LIN {X 0,Y 244.546,Z 349.21,A -85,B 0,C 180,E1 -19754.66,E2 -19754.66} C_VEL
LIN {X 0,Y 242.026,Z 345.394,A -85,B 0,C 180,E1 -19755.456,E2 -19755.456} C_VEL
LIN {X 0,Y 239.218,Z 341.212,A -85,B 0,C 180,E1 -19756.337,E2 -19756.337} C_VEL
LIN {X 0,Y 238.833,Z 340.13,A -85,B 0,C 180,E1 -19756.54,E2 -19756.54} C_VEL
LIN {X 0,Y 238.266,Z 336.796,A -85,B 0,C 180,E1 -19760.076,E2 -19760.076} C_VEL
LIN {X 0,Y 237.671,Z 333.533,A -85,B 0,C 180,E1 -19763.743,E2 -19763.743} C_VEL
LIN {X 0,Y 237.026,Z 330.381,A -85,B 0,C 180,E1 -19767.743,E2 -19767.743} C_VEL
LIN {X 0,Y 236.378,Z 327.428,A -85,B 0,C 180,E1 -19771.594,E2 -19771.594} C_VEL
LIN {X 0,Y 235.759,Z 324.904,A -85,B 0,C 180,E1 -19775.333,E2 -19775.333} C_VEL
LIN {X 0,Y 235.115,Z 322.576,A -85,B 0,C 180,E1 -19778.979,E2 -19778.979} C_VEL
LIN {X 0,Y 234.966,Z 321.838,A -85,B 0,C 180,E1 -19780.336,E2 -19780.336} C_VEL
LIN {X 0,Y 235.086,Z 321.809,A -85,B 0,C 180,E1 -19784.392,E2 -19784.392} C_VEL
LIN {X 0,Y 235.285,Z 321.791,A -85,B 0,C 180,E1 -19790.302,E2 -19790.302} C_VEL
LIN {X 0,Y 235.355,Z 321.768,A -85,B 0,C 180,E1 -19793.14,E2 -19793.14} C_VEL
LIN {X 0,Y 235.594,Z 321.742,A -85,B 0,C 180,E1 -19798.29,E2 -19798.29} C_VEL
LIN {X 0,Y 235.59,Z 321.753,A -85,B 0,C 180,E1 -19801.709,E2 -19801.709} C_VEL
LIN {X 0,Y 235.36,Z 321.774,A -85,B 0,C 180,E1 -19806.86,E2 -19806.86} C_VEL
LIN {X 0,Y 235.213,Z 321.785,A -85,B 0,C 180,E1 -19810.327,E2 -19810.327} C_VEL
LIN {X 0,Y 235.114,Z 321.8,A -85,B 0,C 180,E1 -19815.606,E2 -19815.606} C_VEL
LIN {X 0,Y 235.008,Z 321.838,A -85,B 0,C 180,E1 -19819.205,E2 -19819.205} C_VEL
LIN {X 0,Y 234.981,Z 321.816,A -85,B 0,C 180,E1 -19821.415,E2 -19821.415} C_VEL
LIN {X 0,Y 236.066,Z 324.801,A -85,B 0,C 180,E1 -19824.632,E2 -19824.632} C_VEL
LIN {X 0,Y 237.859,Z 328.745,A -85,B 0,C 180,E1 -19828.213,E2 -19828.213} C_VEL
LIN {X 0,Y 239.119,Z 334.547,A -85,B 0,C 180,E1 -19831.941,E2 -19831.941} C_VEL
LIN {X 0,Y 240.693,Z 341.686,A -85,B 0,C 180,E1 -19835.731,E2 -19835.731} C_VEL
LIN {X 0,Y 241.887,Z 346.106,A -85,B 0,C 180,E1 -19837.864,E2 -19837.864} C_VEL
LIN {X 0,Y 241.737,Z 348.256,A -85,B 0,C 180,E1 -19838.655,E2 -19838.655} C_VEL
LIN {X 0,Y 239.964,Z 352.557,A -85,B 0,C 180,E1 -19839.813,E2 -19839.813} C_VEL
LIN {X 0,Y 238.2,Z 356.932,A -85,B 0,C 180,E1 -19840.981,E2 -19840.981} C_VEL
LIN {X 0,Y 238.102,Z 359.179,A -85,B 0,C 180,E1 -19841.776,E2 -19841.776} C_VEL
LIN {X 0,Y 239.25,Z 364.152,A -85,B 0,C 180,E1 -19843.728,E2 -19843.728} C_VEL
LIN {X 0,Y 243.073,Z 371.351,A -85,B 0,C 180,E1 -19844.94,E2 -19844.94} C_VEL
LIN {X 0,Y 247.925,Z 380.694,A -85,B 0,C 180,E1 -19846.438,E2 -19846.438} C_VEL
LIN {X 0,Y 249.092,Z 383.421,A -85,B 0,C 180,E1 -19846.816,E2 -19846.816} C_VEL
LIN {X 0,Y 251.313,Z 398.131,A -85,B 0,C 180,E1 -19848.228,E2 -19848.228} C_VEL
LIN {X 0,Y 252.197,Z 408.726,A -85,B 0,C 180,E1 -19849.304,E2 -19849.304} C_VEL
LIN {X 0,Y 252.44,Z 423.635,A -85,B 0,C 180,E1 -19850.956,E2 -19850.956} C_VEL
LIN {X 0,Y 251.684,Z 438.58,A -85,B 0,C 180,E1 -19852.854,E2 -19852.854} C_VEL
LIN {X 0,Y 251.019,Z 446.409,A -85,B 0,C 180,E1 -19853.988,E2 -19853.988} C_VEL
LIN {X 0,Y 247.709,Z 458.427,A -85,B 0,C 180,E1 -19855.675,E2 -19855.675} C_VEL
LIN {X 0,Y 243.793,Z 470.661,A -85,B 0,C 180,E1 -19857.771,E2 -19857.771} C_VEL
LIN {X 0,Y 239.831,Z 481.837,A -85,B 0,C 180,E1 -19860.121,E2 -19860.121} C_VEL
LIN {X 0,Y 236.508,Z 491.296,A -85,B 0,C 180,E1 -19862.575,E2 -19862.575} C_VEL
LIN {X 0,Y 233.219,Z 500.599,A -85,B 0,C 180,E1 -19865.522,E2 -19865.522} C_VEL
LIN {X 0,Y 230.515,Z 508.344,A -85,B 0,C 180,E1 -19868.54,E2 -19868.54} C_VEL
LIN {X 0,Y 228.316,Z 515.619,A -85,B 0,C 180,E1 -19872.073,E2 -19872.073} C_VEL
LIN {X 0,Y 226.843,Z 521.367,A -85,B 0,C 180,E1 -19875.65,E2 -19875.65} C_VEL
LIN {X 0,Y 226.164,Z 525.743,A -85,B 0,C 180,E1 -19879.255,E2 -19879.255} C_VEL
LIN {X 0,Y 226.138,Z 528.849,A -85,B 0,C 180,E1 -19882.859,E2 -19882.859} C_VEL
LIN {X 0,Y 226.3,Z 529.944,A -85,B 0,C 180,E1 -19884.654,E2 -19884.654} C_VEL
LIN {X 0,Y 226.587,Z 531.209,A -85,B 0,C 180,E1 -19888.223,E2 -19888.223} C_VEL
LIN {X 0,Y 226.725,Z 531.382,A -85,B 0,C 180,E1 -19890,E2 -19890} C_VEL
LIN {X 0,Y 226.622,Z 531.21,A -85,B 0,C 180,E1 -19891.778,E2 -19891.778} C_VEL
LIN {X 0,Y 226.314,Z 529.932,A -85,B 0,C 180,E1 -19895.346,E2 -19895.346} C_VEL
LIN {X 0,Y 226.106,Z 527.426,A -85,B 0,C 180,E1 -19898.941,E2 -19898.941} C_VEL
LIN {X 0,Y 226.418,Z 523.672,A -85,B 0,C 180,E1 -19902.55,E2 -19902.55} C_VEL
LIN {X 0,Y 227.507,Z 518.609,A -85,B 0,C 180,E1 -19906.143,E2 -19906.143} C_VEL
LIN {X 0,Y 229.307,Z 512.105,A -85,B 0,C 180,E1 -19909.703,E2 -19909.703} C_VEL
LIN {X 0,Y 231.689,Z 505.132,A -85,B 0,C 180,E1 -19912.753,E2 -19912.753} C_VEL
LIN {X 0,Y 234.924,Z 495.818,A -85,B 0,C 180,E1 -19916.026,E2 -19916.026} C_VEL
LIN {X 0,Y 235.788,Z 493.383,A -85,B 0,C 180,E1 -19916.797,E2 -19916.797} C_VEL
LIN {X 0,Y 240.246,Z 486.965,A -85,B 0,C 180,E1 -19919.822,E2 -19919.822} C_VEL
LIN {X 0,Y 246.799,Z 477.953,A -85,B 0,C 180,E1 -19923.242,E2 -19923.242} C_VEL
LIN {X 0,Y 253.752,Z 468.674,A -85,B 0,C 180,E1 -19926.054,E2 -19926.054} C_VEL
LIN {X 0,Y 262.443,Z 456.908,A -85,B 0,C 180,E1 -19928.883,E2 -19928.883} C_VEL
LIN {X 0,Y 269.092,Z 446.423,A -85,B 0,C 180,E1 -19931.26,E2 -19931.26} C_VEL
LIN {X 0,Y 272.912,Z 439.616,A -85,B 0,C 180,E1 -19932.85,E2 -19932.85} C_VEL
LIN {X 0,Y 277.489,Z 430.661,A -85,B 0,C 180,E1 -19935.167,E2 -19935.167} C_VEL
LIN {X 0,Y 278.073,Z 429.482,A -85,B 0,C 180,E1 -19935.494,E2 -19935.494} C_VEL
LIN {X 0,Y 278.422,Z 428.515,A -85,B 0,C 180,E1 -19935.872,E2 -19935.872} C_VEL
LIN {X 0,Y 277.94,Z 425.696,A -85,B 0,C 180,E1 -19938.895,E2 -19938.895} C_VEL
LIN {X 0,Y 277.798,Z 424.783,A -85,B 0,C 180,E1 -19940.767,E2 -19940.767} C_VEL
LIN {X 0,Y 277.569,Z 424.76,A -85,B 0,C 180,E1 -19942.579,E2 -19942.579} C_VEL
LIN {X 0,Y 277.242,Z 425.386,A -85,B 0,C 180,E1 -19944.335,E2 -19944.335} C_VEL
LIN {X 0,Y 276.884,Z 426.593,A -85,B 0,C 180,E1 -19946.054,E2 -19946.054} C_VEL
LIN {X 0,Y 276.518,Z 427.587,A -85,B 0,C 180,E1 -19947.007,E2 -19947.007} C_VEL
LIN {X 0,Y 269.045,Z 435.963,A -85,B 0,C 180,E1 -19949.378,E2 -19949.378} C_VEL
LIN {X 0,Y 261.726,Z 443.197,A -85,B 0,C 180,E1 -19951.971,E2 -19951.971} C_VEL
LIN {X 0,Y 255.021,Z 449.015,A -85,B 0,C 180,E1 -19954.713,E2 -19954.713} C_VEL
LIN {X 0,Y 250.476,Z 452.488,A -85,B 0,C 180,E1 -19956.87,E2 -19956.87} C_VEL
LIN {X 0,Y 245.059,Z 455.968,A -85,B 0,C 180,E1 -19959.871,E2 -19959.871} C_VEL
LIN {X 0,Y 240.418,Z 458.16,A -85,B 0,C 180,E1 -19963.003,E2 -19963.003} C_VEL
LIN {X 0,Y 236.524,Z 459.084,A -85,B 0,C 180,E1 -19966.249,E2 -19966.249} C_VEL
LIN {X 0,Y 233.348,Z 458.745,A -85,B 0,C 180,E1 -19969.589,E2 -19969.589} C_VEL
LIN {X 0,Y 231.091,Z 457,A -85,B 0,C 180,E1 -19973.013,E2 -19973.013} C_VEL
LIN {X 0,Y 230.288,Z 455.599,A -85,B 0,C 180,E1 -19974.747,E2 -19974.747} C_VEL
LIN {X 0,Y 229.131,Z 452.894,A -85,B 0,C 180,E1 -19977.363,E2 -19977.363} C_VEL
LIN {X 0,Y 228.201,Z 447.905,A -85,B 0,C 180,E1 -19980.883,E2 -19980.883} C_VEL
LIN {X 0,Y 227.837,Z 441.307,A -85,B 0,C 180,E1 -19984.423,E2 -19984.423} C_VEL
LIN {X 0,Y 228.28,Z 434.052,A -85,B 0,C 180,E1 -19987.519,E2 -19987.519} C_VEL
LIN {X 0,Y 228.851,Z 426.476,A -85,B 0,C 180,E1 -19990.171,E2 -19990.171} C_VEL
LIN {X 0,Y 229.845,Z 415.862,A -85,B 0,C 180,E1 -19993.258,E2 -19993.258} C_VEL
LIN {X 0,Y 230.966,Z 404.89,A -85,B 0,C 180,E1 -19995.894,E2 -19995.894} C_VEL
LIN {X 0,Y 232.532,Z 391.706,A -85,B 0,C 180,E1 -19998.503,E2 -19998.503} C_VEL
LIN {X 0,Y 234.072,Z 378.213,A -85,B 0,C 180,E1 -20000.658,E2 -20000.658} C_VEL
LIN {X 0,Y 235.39,Z 364.819,A -85,B 0,C 180,E1 -20002.415,E2 -20002.415} C_VEL
LIN {X 0,Y 232.483,Z 351.741,A -85,B 0,C 180,E1 -20004.032,E2 -20004.032} C_VEL
LIN {X 0,Y 228.898,Z 336.137,A -85,B 0,C 180,E1 -20005.639,E2 -20005.639} C_VEL
LIN {X 0,Y 227.541,Z 330.01,A -85,B 0,C 180,E1 -20006.188,E2 -20006.188} C_VEL
LIN {X 0,Y 227.571,Z 329.748,A -85,B 0,C 180,E1 -20006.721,E2 -20006.721} C_VEL
LIN {X 0,Y 229.303,Z 332.171,A -85,B 0,C 180,E1 -20010.886,E2 -20010.886} C_VEL
LIN {X 0,Y 230.489,Z 334.719,A -85,B 0,C 180,E1 -20014.585,E2 -20014.585} C_VEL
LIN {X 0,Y 231.235,Z 337.275,A -85,B 0,C 180,E1 -20017.793,E2 -20017.793} C_VEL
LIN {X 0,Y 231.97,Z 341.024,A -85,B 0,C 180,E1 -20021.881,E2 -20021.881} C_VEL
LIN {X 0,Y 233.763,Z 344.267,A -85,B 0,C 180,E1 -20022.524,E2 -20022.524} C_VEL
LIN {X 0,Y 235.368,Z 346.233,A -85,B 0,C 180,E1 -20023.045,E2 -20023.045} C_VEL
LIN {X 0,Y 237.793,Z 349.953,A -85,B 0,C 180,E1 -20023.874,E2 -20023.874} C_VEL
LIN {X 0,Y 242.755,Z 358.409,A -85,B 0,C 180,E1 -20025.621,E2 -20025.621} C_VEL
LIN {X 0,Y 248.115,Z 370.063,A -85,B 0,C 180,E1 -20027.782,E2 -20027.782} C_VEL
LIN {X 0,Y 252.113,Z 381.073,A -85,B 0,C 180,E1 -20029.741,E2 -20029.741} C_VEL
LIN {X 0,Y 255.191,Z 392.133,A -85,B 0,C 180,E1 -20031.704,E2 -20031.704} C_VEL
LIN {X 0,Y 257.251,Z 402.294,A -85,B 0,C 180,E1 -20033.526,E2 -20033.526} C_VEL
LIN {X 0,Y 254.034,Z 415.547,A -85,B 0,C 180,E1 -20035.207,E2 -20035.207} C_VEL
LIN {X 0,Y 250.103,Z 428.688,A -85,B 0,C 180,E1 -20037.252,E2 -20037.252} C_VEL
LIN {X 0,Y 246.362,Z 440.487,A -85,B 0,C 180,E1 -20039.578,E2 -20039.578} C_VEL
LIN {X 0,Y 242.923,Z 450.385,A -85,B 0,C 180,E1 -20041.957,E2 -20041.957} C_VEL
LIN {X 0,Y 239.203,Z 460.038,A -85,B 0,C 180,E1 -20044.784,E2 -20044.784} C_VEL
LIN {X 0,Y 235.58,Z 469.05,A -85,B 0,C 180,E1 -20048.104,E2 -20048.104} C_VEL
LIN {X 0,Y 232.622,Z 476.301,A -85,B 0,C 180,E1 -20051.504,E2 -20051.504} C_VEL
LIN {X 0,Y 230.364,Z 482.03,A -85,B 0,C 180,E1 -20054.97,E2 -20054.97} C_VEL
LIN {X 0,Y 229.02,Z 485.411,A -85,B 0,C 180,E1 -20057.595,E2 -20057.595} C_VEL
LIN {X 0,Y 227.753,Z 488.843,A -85,B 0,C 180,E1 -20061.124,E2 -20061.124} C_VEL
LIN {X 0,Y 227.057,Z 491.092,A -85,B 0,C 180,E1 -20064.672,E2 -20064.672} C_VEL
LIN {X 0,Y 226.961,Z 491.789,A -85,B 0,C 180,E1 -20066.449,E2 -20066.449} C_VEL
LIN {X 0,Y 226.666,Z 492.384,A -85,B 0,C 180,E1 -20070,E2 -20070} C_VEL
LIN {X 0,Y 226.953,Z 491.821,A -85,B 0,C 180,E1 -20073.55,E2 -20073.55} C_VEL
LIN {X 0,Y 227.261,Z 490.191,A -85,B 0,C 180,E1 -20077.105,E2 -20077.105} C_VEL
LIN {X 0,Y 228.333,Z 487.401,A -85,B 0,C 180,E1 -20080.642,E2 -20080.642} C_VEL
LIN {X 0,Y 229.841,Z 483.407,A -85,B 0,C 180,E1 -20084.159,E2 -20084.159} C_VEL
LIN {X 0,Y 231.982,Z 478.083,A -85,B 0,C 180,E1 -20087.635,E2 -20087.635} C_VEL
LIN {X 0,Y 234.782,Z 471.276,A -85,B 0,C 180,E1 -20091.051,E2 -20091.051} C_VEL
LIN {X 0,Y 237.65,Z 463.981,A -85,B 0,C 180,E1 -20093.992,E2 -20093.992} C_VEL
LIN {X 0,Y 241.154,Z 455.15,A -85,B 0,C 180,E1 -20096.854,E2 -20096.854} C_VEL
LIN {X 0,Y 245.123,Z 444.449,A -85,B 0,C 180,E1 -20099.642,E2 -20099.642} C_VEL
LIN {X 0,Y 248.442,Z 434.239,A -85,B 0,C 180,E1 -20101.849,E2 -20101.849} C_VEL
LIN {X 0,Y 252.125,Z 422.537,A -85,B 0,C 180,E1 -20103.883,E2 -20103.883} C_VEL
LIN {X 0,Y 255.802,Z 408.831,A -85,B 0,C 180,E1 -20105.817,E2 -20105.817} C_VEL
LIN {X 0,Y 257.274,Z 402.679,A -85,B 0,C 180,E1 -20106.549,E2 -20106.549} C_VEL
LIN {X 0,Y 255.565,Z 393.25,A -85,B 0,C 180,E1 -20108.218,E2 -20108.218} C_VEL
LIN {X 0,Y 252.318,Z 381.543,A -85,B 0,C 180,E1 -20110.314,E2 -20110.314} C_VEL
LIN {X 0,Y 247.928,Z 369.544,A -85,B 0,C 180,E1 -20112.461,E2 -20112.461} C_VEL
LIN {X 0,Y 243.36,Z 359.711,A -85,B 0,C 180,E1 -20114.303,E2 -20114.303} C_VEL
LIN {X 0,Y 239.774,Z 353.345,A -85,B 0,C 180,E1 -20115.6,E2 -20115.6} C_VEL
LIN {X 0,Y 236.943,Z 348.944,A -85,B 0,C 180,E1 -20116.563,E2 -20116.563} C_VEL
LIN {X 0,Y 234.611,Z 345.246,A -85,B 0,C 180,E1 -20117.367,E2 -20117.367} C_VEL
LIN {X 0,Y 232.509,Z 342.318,A -85,B 0,C 180,E1 -20118.077,E2 -20118.077} C_VEL
LIN {X 0,Y 231.954,Z 340.941,A -85,B 0,C 180,E1 -20118.339,E2 -20118.339} C_VEL
LIN {X 0,Y 231.249,Z 337.138,A -85,B 0,C 180,E1 -20122.567,E2 -20122.567} C_VEL
LIN {X 0,Y 230.596,Z 333.766,A -85,B 0,C 180,E1 -20126.729,E2 -20126.729} C_VEL
LIN {X 0,Y 229.967,Z 330.832,A -85,B 0,C 180,E1 -20130.727,E2 -20130.727} C_VEL
LIN {X 0,Y 229.364,Z 328.262,A -85,B 0,C 180,E1 -20134.597,E2 -20134.597} C_VEL
LIN {X 0,Y 228.784,Z 325.943,A -85,B 0,C 180,E1 -20138.369,E2 -20138.369} C_VEL
LIN {X 0,Y 228.218,Z 323.635,A -85,B 0,C 180,E1 -20142.677,E2 -20142.677} C_VEL
LIN {X 0,Y 228.048,Z 322.69,A -85,B 0,C 180,E1 -20144.814,E2 -20144.814} C_VEL
LIN {X 0,Y 228.228,Z 322.668,A -85,B 0,C 180,E1 -20150.196,E2 -20150.196} C_VEL
LIN {X 0,Y 228.307,Z 322.647,A -85,B 0,C 180,E1 -20152.927,E2 -20152.927} C_VEL
LIN {X 0,Y 228.552,Z 322.619,A -85,B 0,C 180,E1 -20158.238,E2 -20158.238} C_VEL
LIN {X 0,Y 228.548,Z 322.63,A -85,B 0,C 180,E1 -20161.762,E2 -20161.762} C_VEL
LIN {X 0,Y 228.312,Z 322.654,A -85,B 0,C 180,E1 -20167.073,E2 -20167.073} C_VEL
LIN {X 0,Y 228.144,Z 322.663,A -85,B 0,C 180,E1 -20170.651,E2 -20170.651} C_VEL
LIN {X 0,Y 228.063,Z 322.695,A -85,B 0,C 180,E1 -20174.272,E2 -20174.272} C_VEL
LIN {X 0,Y 228.093,Z 322.862,A -85,B 0,C 180,E1 -20176.931,E2 -20176.931} C_VEL
LIN {X 0,Y 229.341,Z 326.301,A -85,B 0,C 180,E1 -20181.576,E2 -20181.576} C_VEL
LIN {X 0,Y 231.512,Z 331.916,A -85,B 0,C 180,E1 -20187.087,E2 -20187.087} C_VEL
LIN {X 0,Y 232.505,Z 334.244,A -85,B 0,C 180,E1 -20188.923,E2 -20188.923} C_VEL
LIN {X 0,Y 233.723,Z 340.44,A -85,B 0,C 180,E1 -20192.769,E2 -20192.769} C_VEL
LIN {X 0,Y 235.942,Z 349.846,A -85,B 0,C 180,E1 -20197.635,E2 -20197.635} C_VEL
LIN {X 0,Y 238.102,Z 359.179,A -85,B 0,C 180,E1 -20201.776,E2 -20201.776} C_VEL
LIN {X 0,Y 238.61,Z 361.472,A -85,B 0,C 180,E1 -20202.521,E2 -20202.521} C_VEL
LIN {X 0,Y 239.391,Z 365.932,A -85,B 0,C 180,E1 -20203.416,E2 -20203.416} C_VEL
LIN {X 0,Y 240.22,Z 371.048,A -85,B 0,C 180,E1 -20204.106,E2 -20204.106} C_VEL
LIN {X 0,Y 242.48,Z 382.027,A -85,B 0,C 180,E1 -20205.291,E2 -20205.291} C_VEL
LIN {X 0,Y 243.569,Z 385.469,A -85,B 0,C 180,E1 -20205.739,E2 -20205.739} C_VEL
LIN {X 0,Y 244.229,Z 387.974,A -85,B 0,C 180,E1 -20206.044,E2 -20206.044} C_VEL
LIN {X 0,Y 245.99,Z 401.828,A -85,B 0,C 180,E1 -20207.471,E2 -20207.471} C_VEL
LIN {X 0,Y 246.681,Z 414.824,A -85,B 0,C 180,E1 -20208.889,E2 -20208.889} C_VEL
LIN {X 0,Y 246.357,Z 428.871,A -85,B 0,C 180,E1 -20210.572,E2 -20210.572} C_VEL
LIN {X 0,Y 245.322,Z 442.792,A -85,B 0,C 180,E1 -20212.5,E2 -20212.5} C_VEL
LIN {X 0,Y 244.341,Z 449.602,A -85,B 0,C 180,E1 -20213.522,E2 -20213.522} C_VEL
LIN {X 0,Y 240.275,Z 462.535,A -85,B 0,C 180,E1 -20215.479,E2 -20215.479} C_VEL
LIN {X 0,Y 236.285,Z 473.977,A -85,B 0,C 180,E1 -20217.63,E2 -20217.63} C_VEL
LIN {X 0,Y 232.39,Z 484.518,A -85,B 0,C 180,E1 -20220.067,E2 -20220.067} C_VEL
LIN {X 0,Y 229.093,Z 493.486,A -85,B 0,C 180,E1 -20222.603,E2 -20222.603} C_VEL
LIN {X 0,Y 225.834,Z 502.328,A -85,B 0,C 180,E1 -20225.648,E2 -20225.648} C_VEL
LIN {X 0,Y 223.142,Z 509.704,A -85,B 0,C 180,E1 -20228.765,E2 -20228.765} C_VEL
LIN {X 0,Y 221.011,Z 516.467,A -85,B 0,C 180,E1 -20232.343,E2 -20232.343} C_VEL
LIN {X 0,Y 219.624,Z 521.99,A -85,B 0,C 180,E1 -20236.114,E2 -20236.114} C_VEL
LIN {X 0,Y 219.116,Z 525.127,A -85,B 0,C 180,E1 -20238.905,E2 -20238.905} C_VEL
LIN {X 0,Y 219.036,Z 528.234,A -85,B 0,C 180,E1 -20242.627,E2 -20242.627} C_VEL
LIN {X 0,Y 219.218,Z 529.332,A -85,B 0,C 180,E1 -20244.481,E2 -20244.481} C_VEL
LIN {X 0,Y 219.491,Z 530.599,A -85,B 0,C 180,E1 -20248.166,E2 -20248.166} C_VEL
LIN {X 0,Y 219.669,Z 530.775,A -85,B 0,C 180,E1 -20250,E2 -20250} C_VEL
LIN {X 0,Y 219.525,Z 530.599,A -85,B 0,C 180,E1 -20251.835,E2 -20251.835} C_VEL
LIN {X 0,Y 219.23,Z 529.32,A -85,B 0,C 180,E1 -20255.519,E2 -20255.519} C_VEL
LIN {X 0,Y 219.017,Z 526.809,A -85,B 0,C 180,E1 -20259.233,E2 -20259.233} C_VEL
LIN {X 0,Y 219.416,Z 523.055,A -85,B 0,C 180,E1 -20262.957,E2 -20262.957} C_VEL
LIN {X 0,Y 220.578,Z 517.988,A -85,B 0,C 180,E1 -20266.664,E2 -20266.664} C_VEL
LIN {X 0,Y 222.515,Z 511.484,A -85,B 0,C 180,E1 -20270.331,E2 -20270.331} C_VEL
LIN {X 0,Y 225.468,Z 503.374,A -85,B 0,C 180,E1 -20273.905,E2 -20273.905} C_VEL
LIN {X 0,Y 228.946,Z 493.971,A -85,B 0,C 180,E1 -20277.257,E2 -20277.257} C_VEL
LIN {X 0,Y 235.501,Z 485.464,A -85,B 0,C 180,E1 -20281.484,E2 -20281.484} C_VEL
LIN {X 0,Y 242.624,Z 476.611,A -85,B 0,C 180,E1 -20284.897,E2 -20284.897} C_VEL
LIN {X 0,Y 251.076,Z 466.267,A -85,B 0,C 180,E1 -20288.012,E2 -20288.012} C_VEL
LIN {X 0,Y 259.375,Z 455.746,A -85,B 0,C 180,E1 -20290.565,E2 -20290.565} C_VEL
LIN {X 0,Y 266.845,Z 444.669,A -85,B 0,C 180,E1 -20293.218,E2 -20293.218} C_VEL
LIN {X 0,Y 271.904,Z 436.065,A -85,B 0,C 180,E1 -20295.507,E2 -20295.507} C_VEL
LIN {X 0,Y 273.119,Z 434.001,A -85,B 0,C 180,E1 -20296.097,E2 -20296.097} C_VEL
LIN {X 0,Y 273.366,Z 432.541,A -85,B 0,C 180,E1 -20297.06,E2 -20297.06} C_VEL
LIN {X 0,Y 273.043,Z 430.396,A -85,B 0,C 180,E1 -20299.948,E2 -20299.948} C_VEL
LIN {X 0,Y 272.853,Z 429.885,A -85,B 0,C 180,E1 -20301.817,E2 -20301.817} C_VEL
LIN {X 0,Y 272.407,Z 430.234,A -85,B 0,C 180,E1 -20303.602,E2 -20303.602} C_VEL
LIN {X 0,Y 271.801,Z 431.438,A -85,B 0,C 180,E1 -20305.836,E2 -20305.836} C_VEL
LIN {X 0,Y 271.498,Z 431.892,A -85,B 0,C 180,E1 -20306.317,E2 -20306.317} C_VEL
LIN {X 0,Y 263.607,Z 439.776,A -85,B 0,C 180,E1 -20308.676,E2 -20308.676} C_VEL
LIN {X 0,Y 256.054,Z 446.503,A -85,B 0,C 180,E1 -20311.293,E2 -20311.293} C_VEL
LIN {X 0,Y 249.102,Z 451.883,A -85,B 0,C 180,E1 -20314.068,E2 -20314.068} C_VEL
LIN {X 0,Y 244.374,Z 455.032,A -85,B 0,C 180,E1 -20316.258,E2 -20316.258} C_VEL
LIN {X 0,Y 238.718,Z 458.149,A -85,B 0,C 180,E1 -20319.312,E2 -20319.312} C_VEL
LIN {X 0,Y 233.875,Z 459.991,A -85,B 0,C 180,E1 -20322.512,E2 -20322.512} C_VEL
LIN {X 0,Y 229.812,Z 460.584,A -85,B 0,C 180,E1 -20325.839,E2 -20325.839} C_VEL
LIN {X 0,Y 226.479,Z 459.91,A -85,B 0,C 180,E1 -20329.27,E2 -20329.27} C_VEL
LIN {X 0,Y 224.113,Z 457.883,A -85,B 0,C 180,E1 -20332.794,E2 -20332.794} C_VEL
LIN {X 0,Y 223.265,Z 456.353,A -85,B 0,C 180,E1 -20334.581,E2 -20334.581} C_VEL
LIN {X 0,Y 222.066,Z 453.407,A -85,B 0,C 180,E1 -20337.279,E2 -20337.279} C_VEL
LIN {X 0,Y 221.115,Z 448.173,A -85,B 0,C 180,E1 -20340.911,E2 -20340.911} C_VEL
LIN {X 0,Y 220.755,Z 443.149,A -85,B 0,C 180,E1 -20343.651,E2 -20343.651} C_VEL
LIN {X 0,Y 221.03,Z 436.02,A -85,B 0,C 180,E1 -20346.848,E2 -20346.848} C_VEL
LIN {X 0,Y 221.707,Z 427.577,A -85,B 0,C 180,E1 -20349.952,E2 -20349.952} C_VEL
LIN {X 0,Y 222.602,Z 418.327,A -85,B 0,C 180,E1 -20352.768,E2 -20352.768} C_VEL
LIN {X 0,Y 223.632,Z 407.613,A -85,B 0,C 180,E1 -20355.494,E2 -20355.494} C_VEL
LIN {X 0,Y 224.972,Z 395.921,A -85,B 0,C 180,E1 -20357.968,E2 -20357.968} C_VEL
LIN {X 0,Y 226.497,Z 383.255,A -85,B 0,C 180,E1 -20360.194,E2 -20360.194} C_VEL
LIN {X 0,Y 227.81,Z 371.173,A -85,B 0,C 180,E1 -20361.966,E2 -20361.966} C_VEL
LIN {X 0,Y 228.33,Z 366.447,A -85,B 0,C 180,E1 -20362.57,E2 -20362.57} C_VEL
LIN {X 0,Y 226.469,Z 357.043,A -85,B 0,C 180,E1 -20363.793,E2 -20363.793} C_VEL
LIN {X 0,Y 223.005,Z 341.761,A -85,B 0,C 180,E1 -20365.513,E2 -20365.513} C_VEL
LIN {X 0,Y 220.899,Z 332.546,A -85,B 0,C 180,E1 -20366.397,E2 -20366.397} C_VEL
LIN {X 0,Y 222.567,Z 334.617,A -85,B 0,C 180,E1 -20370.347,E2 -20370.347} C_VEL
LIN {X 0,Y 223.878,Z 337.279,A -85,B 0,C 180,E1 -20374.407,E2 -20374.407} C_VEL
LIN {X 0,Y 224.769,Z 340.716,A -85,B 0,C 180,E1 -20378.708,E2 -20378.708} C_VEL
LIN {X 0,Y 225.047,Z 341.87,A -85,B 0,C 180,E1 -20379.88,E2 -20379.88} C_VEL
LIN {X 0,Y 227.024,Z 345.18,A -85,B 0,C 180,E1 -20380.644,E2 -20380.644} C_VEL
LIN {X 0,Y 228.657,Z 347.106,A -85,B 0,C 180,E1 -20381.22,E2 -20381.22} C_VEL
LIN {X 0,Y 231.013,Z 350.662,A -85,B 0,C 180,E1 -20382.094,E2 -20382.094} C_VEL
LIN {X 0,Y 236.606,Z 359.784,A -85,B 0,C 180,E1 -20384.195,E2 -20384.195} C_VEL
LIN {X 0,Y 241.172,Z 369.128,A -85,B 0,C 180,E1 -20386.097,E2 -20386.097} C_VEL
LIN {X 0,Y 246.114,Z 382.366,A -85,B 0,C 180,E1 -20388.618,E2 -20388.618} C_VEL
LIN {X 0,Y 249.392,Z 394.465,A -85,B 0,C 180,E1 -20390.881,E2 -20390.881} C_VEL
LIN {X 0,Y 251.222,Z 404.031,A -85,B 0,C 180,E1 -20392.685,E2 -20392.685} C_VEL
LIN {X 0,Y 248.268,Z 416.145,A -85,B 0,C 180,E1 -20394.277,E2 -20394.277} C_VEL
LIN {X 0,Y 244.186,Z 429.29,A -85,B 0,C 180,E1 -20396.355,E2 -20396.355} C_VEL
LIN {X 0,Y 240.29,Z 441.091,A -85,B 0,C 180,E1 -20398.724,E2 -20398.724} C_VEL
LIN {X 0,Y 236.715,Z 450.989,A -85,B 0,C 180,E1 -20401.153,E2 -20401.153} C_VEL
LIN {X 0,Y 232.822,Z 460.645,A -85,B 0,C 180,E1 -20404.042,E2 -20404.042} C_VEL
LIN {X 0,Y 229.009,Z 469.659,A -85,B 0,C 180,E1 -20407.442,E2 -20407.442} C_VEL
LIN {X 0,Y 225.913,Z 476.91,A -85,B 0,C 180,E1 -20410.934,E2 -20410.934} C_VEL
LIN {X 0,Y 223.539,Z 482.639,A -85,B 0,C 180,E1 -20414.5,E2 -20414.5} C_VEL
LIN {X 0,Y 222.108,Z 486.02,A -85,B 0,C 180,E1 -20417.203,E2 -20417.203} C_VEL
LIN {X 0,Y 220.772,Z 489.451,A -85,B 0,C 180,E1 -20420.841,E2 -20420.841} C_VEL
LIN {X 0,Y 220,Z 491.702,A -85,B 0,C 180,E1 -20424.5,E2 -20424.5} C_VEL
LIN {X 0,Y 219.92,Z 492.396,A -85,B 0,C 180,E1 -20426.335,E2 -20426.335} C_VEL
LIN {X 0,Y 219.618,Z 492.99,A -85,B 0,C 180,E1 -20430,E2 -20430} C_VEL
LIN {X 0,Y 219.891,Z 492.429,A -85,B 0,C 180,E1 -20433.665,E2 -20433.665} C_VEL
LIN {X 0,Y 220.248,Z 490.799,A -85,B 0,C 180,E1 -20437.333,E2 -20437.333} C_VEL
LIN {X 0,Y 221.38,Z 488.008,A -85,B 0,C 180,E1 -20440.98,E2 -20440.98} C_VEL
LIN {X 0,Y 222.984,Z 484.014,A -85,B 0,C 180,E1 -20444.604,E2 -20444.604} C_VEL
LIN {X 0,Y 225.237,Z 478.69,A -85,B 0,C 180,E1 -20448.181,E2 -20448.181} C_VEL
LIN {X 0,Y 228.179,Z 471.882,A -85,B 0,C 180,E1 -20451.691,E2 -20451.691} C_VEL
LIN {X 0,Y 231.185,Z 464.585,A -85,B 0,C 180,E1 -20454.708,E2 -20454.708} C_VEL
LIN {X 0,Y 234.841,Z 455.754,A -85,B 0,C 180,E1 -20457.636,E2 -20457.636} C_VEL
LIN {X 0,Y 238.982,Z 445.05,A -85,B 0,C 180,E1 -20460.483,E2 -20460.483} C_VEL
LIN {X 0,Y 242.386,Z 435.071,A -85,B 0,C 180,E1 -20462.683,E2 -20462.683} C_VEL
LIN {X 0,Y 246.285,Z 423.131,A -85,B 0,C 180,E1 -20464.8,E2 -20464.8} C_VEL
LIN {X 0,Y 250.01,Z 409.813,A -85,B 0,C 180,E1 -20466.714,E2 -20466.714} C_VEL
LIN {X 0,Y 251.323,Z 404.365,A -85,B 0,C 180,E1 -20467.381,E2 -20467.381} C_VEL
LIN {X 0,Y 249.309,Z 393.906,A -85,B 0,C 180,E1 -20469.359,E2 -20469.359} C_VEL
LIN {X 0,Y 246.392,Z 383.239,A -85,B 0,C 180,E1 -20471.371,E2 -20471.371} C_VEL
LIN {X 0,Y 242.015,Z 371.177,A -85,B 0,C 180,E1 -20473.656,E2 -20473.656} C_VEL
LIN {X 0,Y 237.338,Z 361.17,A -85,B 0,C 180,E1 -20475.681,E2 -20475.681} C_VEL
LIN {X 0,Y 232.512,Z 353.174,A -85,B 0,C 180,E1 -20477.511,E2 -20477.511} C_VEL
LIN {X 0,Y 230.662,Z 350.293,A -85,B 0,C 180,E1 -20478.196,E2 -20478.196} C_VEL
LIN {X 0,Y 228.049,Z 346.302,A -85,B 0,C 180,E1 -20479.17,E2 -20479.17} C_VEL
LIN {X 0,Y 225.675,Z 343.232,A -85,B 0,C 180,E1 -20480.036,E2 -20480.036} C_VEL
LIN {X 0,Y 224.994,Z 341.744,A -85,B 0,C 180,E1 -20480.328,E2 -20480.328} C_VEL
LIN {X 0,Y 224.351,Z 338.252,A -85,B 0,C 180,E1 -20484.535,E2 -20484.535} C_VEL
LIN {X 0,Y 223.829,Z 335.627,A -85,B 0,C 180,E1 -20487.97,E2 -20487.97} C_VEL
LIN {X 0,Y 223.277,Z 332.957,A -85,B 0,C 180,E1 -20491.826,E2 -20491.826} C_VEL
LIN {X 0,Y 222.658,Z 330.172,A -85,B 0,C 180,E1 -20496.256,E2 -20496.256} C_VEL
LIN {X 0,Y 222.245,Z 328.332,A -85,B 0,C 180,E1 -20499.644,E2 -20499.644} C_VEL
LIN {X 0,Y 221.806,Z 326.469,A -85,B 0,C 180,E1 -20503.431,E2 -20503.431} C_VEL
LIN {X 0,Y 221.317,Z 324.943,A -85,B 0,C 180,E1 -20507.156,E2 -20507.156} C_VEL
LIN {X 0,Y 221.218,Z 323.554,A -85,B 0,C 180,E1 -20511.32,E2 -20511.32} C_VEL
LIN {X 0,Y 221.124,Z 323.538,A -85,B 0,C 180,E1 -20514.528,E2 -20514.528} C_VEL
LIN {X 0,Y 221.51,Z 323.496,A -85,B 0,C 180,E1 -20518.182,E2 -20518.182} C_VEL
LIN {X 0,Y 221.505,Z 323.508,A -85,B 0,C 180,E1 -20521.818,E2 -20521.818} C_VEL
LIN {X 0,Y 221.248,Z 323.536,A -85,B 0,C 180,E1 -20527.3,E2 -20527.3} C_VEL
LIN {X 0,Y 221.193,Z 323.749,A -85,B 0,C 180,E1 -20529.948,E2 -20529.948} C_VEL
LIN {X 0,Y 222.334,Z 326.831,A -85,B 0,C 180,E1 -20536.528,E2 -20536.528} C_VEL
LIN {X 0,Y 223.792,Z 331.117,A -85,B 0,C 180,E1 -20542.139,E2 -20542.139} C_VEL
LIN {X 0,Y 226.323,Z 336.955,A -85,B 0,C 180,E1 -20547.761,E2 -20547.761} C_VEL
LIN {X 0,Y 227.308,Z 341.281,A -85,B 0,C 180,E1 -20550.673,E2 -20550.673} C_VEL
LIN {X 0,Y 228.667,Z 348.192,A -85,B 0,C 180,E1 -20554.651,E2 -20554.651} C_VEL
LIN {X 0,Y 230.529,Z 356.219,A -85,B 0,C 180,E1 -20558.68,E2 -20558.68} C_VEL
LIN {X 0,Y 232.118,Z 363.344,A -85,B 0,C 180,E1 -20561.849,E2 -20561.849} C_VEL
LIN {X 0,Y 234.956,Z 368.554,A -85,B 0,C 180,E1 -20562.832,E2 -20562.832} C_VEL
LIN {X 0,Y 238.943,Z 376.142,A -85,B 0,C 180,E1 -20564.164,E2 -20564.164} C_VEL
LIN {X 0,Y 243.569,Z 385.469,A -85,B 0,C 180,E1 -20565.739,E2 -20565.739} C_VEL
LIN {X 0,Y 244.403,Z 388.882,A -85,B 0,C 180,E1 -20566.14,E2 -20566.14} C_VEL
LIN {X 0,Y 244.629,Z 392.582,A -85,B 0,C 180,E1 -20566.438,E2 -20566.438} C_VEL
LIN {X 0,Y 243.665,Z 400.287,A -85,B 0,C 180,E1 -20566.848,E2 -20566.848} C_VEL
LIN {X 0,Y 241.557,Z 410.073,A -85,B 0,C 180,E1 -20567.35,E2 -20567.35} C_VEL
LIN {X 0,Y 240.98,Z 415.692,A -85,B 0,C 180,E1 -20567.876,E2 -20567.876} C_VEL
LIN {X 0,Y 240.516,Z 429.637,A -85,B 0,C 180,E1 -20569.619,E2 -20569.619} C_VEL
LIN {X 0,Y 239.245,Z 443.707,A -85,B 0,C 180,E1 -20571.643,E2 -20571.643} C_VEL
LIN {X 0,Y 238.447,Z 449.497,A -85,B 0,C 180,E1 -20572.56,E2 -20572.56} C_VEL
LIN {X 0,Y 234.427,Z 461.935,A -85,B 0,C 180,E1 -20574.49,E2 -20574.49} C_VEL
LIN {X 0,Y 230.293,Z 473.374,A -85,B 0,C 180,E1 -20576.68,E2 -20576.68} C_VEL
LIN {X 0,Y 226.203,Z 483.91,A -85,B 0,C 180,E1 -20579.16,E2 -20579.16} C_VEL
LIN {X 0,Y 222.724,Z 492.873,A -85,B 0,C 180,E1 -20581.75,E2 -20581.75} C_VEL
LIN {X 0,Y 219.263,Z 501.71,A -85,B 0,C 180,E1 -20584.869,E2 -20584.869} C_VEL
LIN {X 0,Y 216.445,Z 509.088,A -85,B 0,C 180,E1 -20588.075,E2 -20588.075} C_VEL
LIN {X 0,Y 214.088,Z 516.071,A -85,B 0,C 180,E1 -20591.902,E2 -20591.902} C_VEL
LIN {X 0,Y 212.638,Z 521.372,A -85,B 0,C 180,E1 -20595.648,E2 -20595.648} C_VEL
LIN {X 0,Y 212.087,Z 524.512,A -85,B 0,C 180,E1 -20598.532,E2 -20598.532} C_VEL
LIN {X 0,Y 211.944,Z 527.619,A -85,B 0,C 180,E1 -20602.378,E2 -20602.378} C_VEL
LIN {X 0,Y 212.146,Z 528.721,A -85,B 0,C 180,E1 -20604.297,E2 -20604.297} C_VEL
LIN {X 0,Y 212.396,Z 529.988,A -85,B 0,C 180,E1 -20608.104,E2 -20608.104} C_VEL
LIN {X 0,Y 212.613,Z 530.168,A -85,B 0,C 180,E1 -20610,E2 -20610} C_VEL
LIN {X 0,Y 212.429,Z 529.989,A -85,B 0,C 180,E1 -20611.896,E2 -20611.896} C_VEL
LIN {X 0,Y 212.111,Z 528.441,A -85,B 0,C 180,E1 -20616.278,E2 -20616.278} C_VEL
LIN {X 0,Y 211.952,Z 526.193,A -85,B 0,C 180,E1 -20619.544,E2 -20619.544} C_VEL
LIN {X 0,Y 212.424,Z 522.437,A -85,B 0,C 180,E1 -20623.391,E2 -20623.391} C_VEL
LIN {X 0,Y 213.681,Z 517.368,A -85,B 0,C 180,E1 -20627.219,E2 -20627.219} C_VEL
LIN {X 0,Y 215.772,Z 510.865,A -85,B 0,C 180,E1 -20630.995,E2 -20630.995} C_VEL
LIN {X 0,Y 218.916,Z 502.757,A -85,B 0,C 180,E1 -20634.668,E2 -20634.668} C_VEL
LIN {X 0,Y 222.194,Z 494.319,A -85,B 0,C 180,E1 -20637.804,E2 -20637.804} C_VEL
LIN {X 0,Y 227.999,Z 487.476,A -85,B 0,C 180,E1 -20641.603,E2 -20641.603} C_VEL
LIN {X 0,Y 234.225,Z 480.347,A -85,B 0,C 180,E1 -20644.758,E2 -20644.758} C_VEL
LIN {X 0,Y 242.57,Z 471.068,A -85,B 0,C 180,E1 -20648.002,E2 -20648.002} C_VEL
LIN {X 0,Y 251.338,Z 461.172,A -85,B 0,C 180,E1 -20650.714,E2 -20650.714} C_VEL
LIN {X 0,Y 257.183,Z 453.908,A -85,B 0,C 180,E1 -20652.531,E2 -20652.531} C_VEL
LIN {X 0,Y 262.064,Z 447.255,A -85,B 0,C 180,E1 -20654.209,E2 -20654.209} C_VEL
LIN {X 0,Y 267.109,Z 439.743,A -85,B 0,C 180,E1 -20656.318,E2 -20656.318} C_VEL
LIN {X 0,Y 268.269,Z 437.591,A -85,B 0,C 180,E1 -20657.184,E2 -20657.184} C_VEL
LIN {X 0,Y 268.04,Z 435.753,A -85,B 0,C 180,E1 -20659.498,E2 -20659.498} C_VEL
LIN {X 0,Y 267.93,Z 435.044,A -85,B 0,C 180,E1 -20660.984,E2 -20660.984} C_VEL
LIN {X 0,Y 267.515,Z 434.99,A -85,B 0,C 180,E1 -20662.826,E2 -20662.826} C_VEL
LIN {X 0,Y 266.802,Z 435.668,A -85,B 0,C 180,E1 -20664.746,E2 -20664.746} C_VEL
LIN {X 0,Y 266.128,Z 436.519,A -85,B 0,C 180,E1 -20665.673,E2 -20665.673} C_VEL
LIN {X 0,Y 258.477,Z 443.357,A -85,B 0,C 180,E1 -20667.87,E2 -20667.87} C_VEL
LIN {X 0,Y 250.392,Z 449.745,A -85,B 0,C 180,E1 -20670.581,E2 -20670.581} C_VEL
LIN {X 0,Y 243.19,Z 454.657,A -85,B 0,C 180,E1 -20673.389,E2 -20673.389} C_VEL
LIN {X 0,Y 238.276,Z 457.514,A -85,B 0,C 180,E1 -20675.611,E2 -20675.611} C_VEL
LIN {X 0,Y 232.386,Z 460.245,A -85,B 0,C 180,E1 -20678.721,E2 -20678.721} C_VEL
LIN {X 0,Y 227.32,Z 461.745,A -85,B 0,C 180,E1 -20681.991,E2 -20681.991} C_VEL
LIN {X 0,Y 223.094,Z 462.014,A -85,B 0,C 180,E1 -20685.403,E2 -20685.403} C_VEL
LIN {X 0,Y 219.614,Z 461.05,A -85,B 0,C 180,E1 -20688.93,E2 -20688.93} C_VEL
LIN {X 0,Y 217.138,Z 458.733,A -85,B 0,C 180,E1 -20692.561,E2 -20692.561} C_VEL
LIN {X 0,Y 215.746,Z 456.076,A -85,B 0,C 180,E1 -20695.329,E2 -20695.329} C_VEL
LIN {X 0,Y 214.428,Z 451.314,A -85,B 0,C 180,E1 -20699.061,E2 -20699.061} C_VEL
LIN {X 0,Y 213.758,Z 444.941,A -85,B 0,C 180,E1 -20702.827,E2 -20702.827} C_VEL
LIN {X 0,Y 213.834,Z 437.962,A -85,B 0,C 180,E1 -20706.132,E2 -20706.132} C_VEL
LIN {X 0,Y 214.512,Z 429.43,A -85,B 0,C 180,E1 -20709.429,E2 -20709.429} C_VEL
LIN {X 0,Y 215.473,Z 419.029,A -85,B 0,C 180,E1 -20712.719,E2 -20712.719} C_VEL
LIN {X 0,Y 216.512,Z 408.36,A -85,B 0,C 180,E1 -20715.533,E2 -20715.533} C_VEL
LIN {X 0,Y 217.869,Z 396.602,A -85,B 0,C 180,E1 -20718.089,E2 -20718.089} C_VEL
LIN {X 0,Y 219.572,Z 382.495,A -85,B 0,C 180,E1 -20720.615,E2 -20720.615} C_VEL
LIN {X 0,Y 221.059,Z 368.892,A -85,B 0,C 180,E1 -20722.59,E2 -20722.59} C_VEL
LIN {X 0,Y 221.265,Z 366.47,A -85,B 0,C 180,E1 -20722.908,E2 -20722.908} C_VEL
LIN {X 0,Y 218.194,Z 352.282,A -85,B 0,C 180,E1 -20724.755,E2 -20724.755} C_VEL
LIN {X 0,Y 214.648,Z 336.572,A -85,B 0,C 180,E1 -20726.454,E2 -20726.454} C_VEL
LIN {X 0,Y 214.46,Z 335.628,A -85,B 0,C 180,E1 -20726.584,E2 -20726.584} C_VEL
LIN {X 0,Y 215.636,Z 336.934,A -85,B 0,C 180,E1 -20729.267,E2 -20729.267} C_VEL
LIN {X 0,Y 216.777,Z 338.862,A -85,B 0,C 180,E1 -20732.548,E2 -20732.548} C_VEL
LIN {X 0,Y 217.719,Z 341.399,A -85,B 0,C 180,E1 -20736.195,E2 -20736.195} C_VEL
LIN {X 0,Y 218.052,Z 342.724,A -85,B 0,C 180,E1 -20737.629,E2 -20737.629} C_VEL
LIN {X 0,Y 220.019,Z 345.874,A -85,B 0,C 180,E1 -20738.465,E2 -20738.465} C_VEL
LIN {X 0,Y 221.969,Z 348.076,A -85,B 0,C 180,E1 -20739.221,E2 -20739.221} C_VEL
LIN {X 0,Y 224.585,Z 351.814,A -85,B 0,C 180,E1 -20740.271,E2 -20740.271} C_VEL
LIN {X 0,Y 228.471,Z 358.016,A -85,B 0,C 180,E1 -20741.846,E2 -20741.846} C_VEL
LIN {X 0,Y 232.704,Z 365.386,A -85,B 0,C 180,E1 -20743.626,E2 -20743.626} C_VEL
LIN {X 0,Y 236.401,Z 373.414,A -85,B 0,C 180,E1 -20745.362,E2 -20745.362} C_VEL
LIN {X 0,Y 240.435,Z 384.691,A -85,B 0,C 180,E1 -20747.629,E2 -20747.629} C_VEL
LIN {X 0,Y 243.587,Z 396.764,A -85,B 0,C 180,E1 -20750.001,E2 -20750.001} C_VEL
LIN {X 0,Y 245.166,Z 405.313,A -85,B 0,C 180,E1 -20751.71,E2 -20751.71} C_VEL
LIN {X 0,Y 245.176,Z 406.844,A -85,B 0,C 180,E1 -20751.979,E2 -20751.979} C_VEL
LIN {X 0,Y 241.433,Z 420.533,A -85,B 0,C 180,E1 -20753.88,E2 -20753.88} C_VEL
LIN {X 0,Y 237.619,Z 431.972,A -85,B 0,C 180,E1 -20755.808,E2 -20755.808} C_VEL
LIN {X 0,Y 233.626,Z 443.427,A -85,B 0,C 180,E1 -20758.234,E2 -20758.234} C_VEL
LIN {X 0,Y 229.902,Z 453.053,A -85,B 0,C 180,E1 -20760.717,E2 -20760.717} C_VEL
LIN {X 0,Y 225.93,Z 462.455,A -85,B 0,C 180,E1 -20763.686,E2 -20763.686} C_VEL
LIN {X 0,Y 222.228,Z 470.814,A -85,B 0,C 180,E1 -20766.989,E2 -20766.989} C_VEL
LIN {X 0,Y 219.231,Z 477.519,A -85,B 0,C 180,E1 -20770.329,E2 -20770.329} C_VEL
LIN {X 0,Y 216.714,Z 483.249,A -85,B 0,C 180,E1 -20773.999,E2 -20773.999} C_VEL
LIN {X 0,Y 215.218,Z 486.628,A -85,B 0,C 180,E1 -20776.786,E2 -20776.786} C_VEL
LIN {X 0,Y 213.789,Z 490.06,A -85,B 0,C 180,E1 -20780.539,E2 -20780.539} C_VEL
LIN {X 0,Y 212.946,Z 492.312,A -85,B 0,C 180,E1 -20784.317,E2 -20784.317} C_VEL
LIN {X 0,Y 212.858,Z 493.005,A -85,B 0,C 180,E1 -20786.213,E2 -20786.213} C_VEL
LIN {X 0,Y 212.57,Z 493.597,A -85,B 0,C 180,E1 -20790,E2 -20790} C_VEL
LIN {X 0,Y 212.832,Z 493.037,A -85,B 0,C 180,E1 -20793.786,E2 -20793.786} C_VEL
LIN {X 0,Y 213.24,Z 491.406,A -85,B 0,C 180,E1 -20797.575,E2 -20797.575} C_VEL
LIN {X 0,Y 214.418,Z 488.618,A -85,B 0,C 180,E1 -20801.341,E2 -20801.341} C_VEL
LIN {X 0,Y 216.145,Z 484.621,A -85,B 0,C 180,E1 -20805.077,E2 -20805.077} C_VEL
LIN {X 0,Y 218.519,Z 479.296,A -85,B 0,C 180,E1 -20808.761,E2 -20808.761} C_VEL
LIN {X 0,Y 221.597,Z 472.489,A -85,B 0,C 180,E1 -20812.369,E2 -20812.369} C_VEL
LIN {X 0,Y 224.78,Z 465.188,A -85,B 0,C 180,E1 -20815.461,E2 -20815.461} C_VEL
LIN {X 0,Y 228.591,Z 456.356,A -85,B 0,C 180,E1 -20818.46,E2 -20818.46} C_VEL
LIN {X 0,Y 232.899,Z 445.65,A -85,B 0,C 180,E1 -20821.368,E2 -20821.368} C_VEL
LIN {X 0,Y 236.359,Z 435.946,A -85,B 0,C 180,E1 -20823.551,E2 -20823.551} C_VEL
LIN {X 0,Y 240.527,Z 423.722,A -85,B 0,C 180,E1 -20825.759,E2 -20825.759} C_VEL
LIN {X 0,Y 244.053,Z 411.641,A -85,B 0,C 180,E1 -20827.533,E2 -20827.533} C_VEL
LIN {X 0,Y 245.344,Z 406.042,A -85,B 0,C 180,E1 -20828.272,E2 -20828.272} C_VEL
LIN {X 0,Y 243.527,Z 396.089,A -85,B 0,C 180,E1 -20830.257,E2 -20830.257} C_VEL
LIN {X 0,Y 240.256,Z 383.964,A -85,B 0,C 180,E1 -20832.665,E2 -20832.665} C_VEL
LIN {X 0,Y 236.088,Z 372.631,A -85,B 0,C 180,E1 -20834.961,E2 -20834.961} C_VEL
LIN {X 0,Y 231.918,Z 363.87,A -85,B 0,C 180,E1 -20836.894,E2 -20836.894} C_VEL
LIN {X 0,Y 226.832,Z 355.403,A -85,B 0,C 180,E1 -20839.003,E2 -20839.003} C_VEL
LIN {X 0,Y 224.265,Z 351.475,A -85,B 0,C 180,E1 -20840.027,E2 -20840.027} C_VEL
LIN {X 0,Y 221.309,Z 347.205,A -85,B 0,C 180,E1 -20841.222,E2 -20841.222} C_VEL
LIN {X 0,Y 218.796,Z 344.128,A -85,B 0,C 180,E1 -20842.227,E2 -20842.227} C_VEL
LIN {X 0,Y 218.046,Z 342.538,A -85,B 0,C 180,E1 -20842.612,E2 -20842.612} C_VEL
LIN {X 0,Y 217.423,Z 339.001,A -85,B 0,C 180,E1 -20847.185,E2 -20847.185} C_VEL
LIN {X 0,Y 216.888,Z 336.39,A -85,B 0,C 180,E1 -20851.033,E2 -20851.033} C_VEL
LIN {X 0,Y 216.328,Z 333.709,A -85,B 0,C 180,E1 -20855.457,E2 -20855.457} C_VEL
LIN {X 0,Y 215.922,Z 331.806,A -85,B 0,C 180,E1 -20859.02,E2 -20859.02} C_VEL
LIN {X 0,Y 215.529,Z 329.977,A -85,B 0,C 180,E1 -20862.934,E2 -20862.934} C_VEL
LIN {X 0,Y 215.16,Z 328.508,A -85,B 0,C 180,E1 -20866.782,E2 -20866.782} C_VEL
LIN {X 0,Y 215.088,Z 327.274,A -85,B 0,C 180,E1 -20870.597,E2 -20870.597} C_VEL
LIN {X 0,Y 214.689,Z 326.503,A -85,B 0,C 180,E1 -20874.364,E2 -20874.364} C_VEL
LIN {X 0,Y 214.847,Z 325.983,A -85,B 0,C 180,E1 -20878.125,E2 -20878.125} C_VEL
LIN {X 0,Y 214.875,Z 325.819,A -85,B 0,C 180,E1 -20880,E2 -20880} C_VEL
LIN {X 0,Y 214.787,Z 325.881,A -85,B 0,C 180,E1 -20881.875,E2 -20881.875} C_VEL
LIN {X 0,Y 215.017,Z 326.968,A -85,B 0,C 180,E1 -20887.512,E2 -20887.512} C_VEL
LIN {X 0,Y 215.306,Z 327.504,A -85,B 0,C 180,E1 -20889.393,E2 -20889.393} C_VEL
LIN {X 0,Y 216.07,Z 330.203,A -85,B 0,C 180,E1 -20895.082,E2 -20895.082} C_VEL
LIN {X 0,Y 216.606,Z 331.317,A -85,B 0,C 180,E1 -20896.978,E2 -20896.978} C_VEL
LIN {X 0,Y 217.567,Z 334.243,A -85,B 0,C 180,E1 -20900.813,E2 -20900.813} C_VEL
LIN {X 0,Y 219.07,Z 337.849,A -85,B 0,C 180,E1 -20904.648,E2 -20904.648} C_VEL
LIN {X 0,Y 220.491,Z 340.955,A -85,B 0,C 180,E1 -20907.527,E2 -20907.527} C_VEL
LIN {X 0,Y 221.652,Z 346.25,A -85,B 0,C 180,E1 -20911.119,E2 -20911.119} C_VEL
LIN {X 0,Y 223.199,Z 354.138,A -85,B 0,C 180,E1 -20915.627,E2 -20915.627} C_VEL
LIN {X 0,Y 224.767,Z 361.458,A -85,B 0,C 180,E1 -20919.285,E2 -20919.285} C_VEL
LIN {X 0,Y 225.059,Z 362.684,A -85,B 0,C 180,E1 -20919.804,E2 -20919.804} C_VEL
LIN {X 0,Y 227.935,Z 367.79,A -85,B 0,C 180,E1 -20920.888,E2 -20920.888} C_VEL
LIN {X 0,Y 234.353,Z 379.989,A -85,B 0,C 180,E1 -20923.227,E2 -20923.227} C_VEL
LIN {X 0,Y 238.986,Z 389.825,A -85,B 0,C 180,E1 -20924.978,E2 -20924.978} C_VEL
LIN {X 0,Y 240.494,Z 403.114,A -85,B 0,C 180,E1 -20926.435,E2 -20926.435} C_VEL
LIN {X 0,Y 240.98,Z 415.692,A -85,B 0,C 180,E1 -20927.876,E2 -20927.876} C_VEL
LIN {X 0,Y 240.41,Z 421.191,A -85,B 0,C 180,E1 -20928.436,E2 -20928.436} C_VEL
LIN {X 0,Y 237.647,Z 430.207,A -85,B 0,C 180,E1 -20929.165,E2 -20929.165} C_VEL
LIN {X 0,Y 234.493,Z 438.991,A -85,B 0,C 180,E1 -20929.971,E2 -20929.971} C_VEL
LIN {X 0,Y 233.289,Z 444.039,A -85,B 0,C 180,E1 -20930.659,E2 -20930.659} C_VEL
LIN {X 0,Y 232.384,Z 450.245,A -85,B 0,C 180,E1 -20931.687,E2 -20931.687} C_VEL
LIN {X 0,Y 228.217,Z 462.466,A -85,B 0,C 180,E1 -20933.644,E2 -20933.644} C_VEL
LIN {X 0,Y 223.563,Z 474.662,A -85,B 0,C 180,E1 -20936.083,E2 -20936.083} C_VEL
LIN {X 0,Y 219.398,Z 484.934,A -85,B 0,C 180,E1 -20938.632,E2 -20938.632} C_VEL
LIN {X 0,Y 215.092,Z 495.441,A -85,B 0,C 180,E1 -20941.909,E2 -20941.909} C_VEL
LIN {X 0,Y 211.443,Z 504.439,A -85,B 0,C 180,E1 -20945.451,E2 -20945.451} C_VEL
LIN {X 0,Y 208.404,Z 512.1,A -85,B 0,C 180,E1 -20949.263,E2 -20949.263} C_VEL
LIN {X 0,Y 206.374,Z 518.224,A -85,B 0,C 180,E1 -20953.174,E2 -20953.174} C_VEL
LIN {X 0,Y 205.194,Z 522.952,A -85,B 0,C 180,E1 -20957.137,E2 -20957.137} C_VEL
LIN {X 0,Y 204.859,Z 525.603,A -85,B 0,C 180,E1 -20960.123,E2 -20960.123} C_VEL
LIN {X 0,Y 205.034,Z 528.107,A -85,B 0,C 180,E1 -20964.098,E2 -20964.098} C_VEL
LIN {X 0,Y 205.302,Z 529.378,A -85,B 0,C 180,E1 -20968.039,E2 -20968.039} C_VEL
LIN {X 0,Y 205.557,Z 529.561,A -85,B 0,C 180,E1 -20970,E2 -20970} C_VEL
LIN {X 0,Y 205.136,Z 528.884,A -85,B 0,C 180,E1 -20973.929,E2 -20973.929} C_VEL
LIN {X 0,Y 205.027,Z 527.944,A -85,B 0,C 180,E1 -20976.243,E2 -20976.243} C_VEL
LIN {X 0,Y 204.875,Z 525.575,A -85,B 0,C 180,E1 -20979.877,E2 -20979.877} C_VEL
LIN {X 0,Y 205.446,Z 521.819,A -85,B 0,C 180,E1 -20983.855,E2 -20983.855} C_VEL
LIN {X 0,Y 206.918,Z 516.452,A -85,B 0,C 180,E1 -20988.007,E2 -20988.007} C_VEL
LIN {X 0,Y 209.043,Z 510.244,A -85,B 0,C 180,E1 -20991.705,E2 -20991.705} C_VEL
LIN {X 0,Y 212.377,Z 502.137,A -85,B 0,C 180,E1 -20995.481,E2 -20995.481} C_VEL
LIN {X 0,Y 215.507,Z 494.555,A -85,B 0,C 180,E1 -20998.407,E2 -20998.407} C_VEL
LIN {X 0,Y 221.964,Z 487.669,A -85,B 0,C 180,E1 -21002.566,E2 -21002.566} C_VEL
LIN {X 0,Y 228.447,Z 480.961,A -85,B 0,C 180,E1 -21005.77,E2 -21005.77} C_VEL
LIN {X 0,Y 237.09,Z 472.202,A -85,B 0,C 180,E1 -21009.044,E2 -21009.044} C_VEL
LIN {X 0,Y 247.912,Z 460.962,A -85,B 0,C 180,E1 -21012.258,E2 -21012.258} C_VEL
LIN {X 0,Y 256.381,Z 450.987,A -85,B 0,C 180,E1 -21014.9,E2 -21014.9} C_VEL
LIN {X 0,Y 261.776,Z 443.923,A -85,B 0,C 180,E1 -21016.948,E2 -21016.948} C_VEL
LIN {X 0,Y 262.481,Z 442.924,A -85,B 0,C 180,E1 -21017.274,E2 -21017.274} C_VEL
LIN {X 0,Y 262.943,Z 441.746,A -85,B 0,C 180,E1 -21018.072,E2 -21018.072} C_VEL
LIN {X 0,Y 262.756,Z 439.96,A -85,B 0,C 180,E1 -21020.866,E2 -21020.866} C_VEL
LIN {X 0,Y 262.548,Z 439.742,A -85,B 0,C 180,E1 -21021.999,E2 -21021.999} C_VEL
LIN {X 0,Y 261.436,Z 440.348,A -85,B 0,C 180,E1 -21024.591,E2 -21024.591} C_VEL
LIN {X 0,Y 259.416,Z 442.054,A -85,B 0,C 180,E1 -21025.325,E2 -21025.325} C_VEL
LIN {X 0,Y 250.768,Z 448.772,A -85,B 0,C 180,E1 -21027.826,E2 -21027.826} C_VEL
LIN {X 0,Y 242.838,Z 454.141,A -85,B 0,C 180,E1 -21030.528,E2 -21030.528} C_VEL
LIN {X 0,Y 235.553,Z 458.324,A -85,B 0,C 180,E1 -21033.414,E2 -21033.414} C_VEL
LIN {X 0,Y 229.028,Z 461.294,A -85,B 0,C 180,E1 -21036.49,E2 -21036.49} C_VEL
LIN {X 0,Y 223.343,Z 463.047,A -85,B 0,C 180,E1 -21039.749,E2 -21039.749} C_VEL
LIN {X 0,Y 218.466,Z 463.596,A -85,B 0,C 180,E1 -21043.171,E2 -21043.171} C_VEL
LIN {X 0,Y 214.403,Z 462.919,A -85,B 0,C 180,E1 -21046.735,E2 -21046.735} C_VEL
LIN {X 0,Y 211.333,Z 460.94,A -85,B 0,C 180,E1 -21050.429,E2 -21050.429} C_VEL
LIN {X 0,Y 209.212,Z 457.631,A -85,B 0,C 180,E1 -21054.216,E2 -21054.216} C_VEL
LIN {X 0,Y 207.694,Z 452.947,A -85,B 0,C 180,E1 -21058.061,E2 -21058.061} C_VEL
LIN {X 0,Y 206.949,Z 448.404,A -85,B 0,C 180,E1 -21060.973,E2 -21060.973} C_VEL
LIN {X 0,Y 206.629,Z 440.895,A -85,B 0,C 180,E1 -21064.878,E2 -21064.878} C_VEL
LIN {X 0,Y 207.269,Z 431.667,A -85,B 0,C 180,E1 -21068.709,E2 -21068.709} C_VEL
LIN {X 0,Y 207.98,Z 422.876,A -85,B 0,C 180,E1 -21071.698,E2 -21071.698} C_VEL
LIN {X 0,Y 209.027,Z 412.699,A -85,B 0,C 180,E1 -21074.606,E2 -21074.606} C_VEL
LIN {X 0,Y 210.337,Z 400.546,A -85,B 0,C 180,E1 -21077.501,E2 -21077.501} C_VEL
LIN {X 0,Y 212.042,Z 387.237,A -85,B 0,C 180,E1 -21080.113,E2 -21080.113} C_VEL
LIN {X 0,Y 213.764,Z 372.331,A -85,B 0,C 180,E1 -21082.47,E2 -21082.47} C_VEL
LIN {X 0,Y 214.155,Z 366.744,A -85,B 0,C 180,E1 -21083.235,E2 -21083.235} C_VEL
LIN {X 0,Y 210.801,Z 351.534,A -85,B 0,C 180,E1 -21085.265,E2 -21085.265} C_VEL
LIN {X 0,Y 207.982,Z 338.812,A -85,B 0,C 180,E1 -21086.734,E2 -21086.734} C_VEL
LIN {X 0,Y 208.357,Z 338.853,A -85,B 0,C 180,E1 -21087.088,E2 -21087.088} C_VEL
LIN {X 0,Y 209.511,Z 340.383,A -85,B 0,C 180,E1 -21090.21,E2 -21090.21} C_VEL
LIN {X 0,Y 210.555,Z 342.305,A -85,B 0,C 180,E1 -21093.439,E2 -21093.439} C_VEL
LIN {X 0,Y 211.006,Z 343.514,A -85,B 0,C 180,E1 -21095.068,E2 -21095.068} C_VEL
LIN {X 0,Y 213.344,Z 347.051,A -85,B 0,C 180,E1 -21096.171,E2 -21096.171} C_VEL
LIN {X 0,Y 215.14,Z 348.959,A -85,B 0,C 180,E1 -21096.94,E2 -21096.94} C_VEL
LIN {X 0,Y 217.819,Z 352.693,A -85,B 0,C 180,E1 -21098.127,E2 -21098.127} C_VEL
LIN {X 0,Y 219.51,Z 355.193,A -85,B 0,C 180,E1 -21098.864,E2 -21098.864} C_VEL
LIN {X 0,Y 222.092,Z 359.086,A -85,B 0,C 180,E1 -21100,E2 -21100} C_VEL
LIN {X 0,Y 226.682,Z 366.856,A -85,B 0,C 180,E1 -21102.078,E2 -21102.078} C_VEL
LIN {X 0,Y 230.597,Z 375.02,A -85,B 0,C 180,E1 -21104.022,E2 -21104.022} C_VEL
LIN {X 0,Y 234.092,Z 384.715,A -85,B 0,C 180,E1 -21106.099,E2 -21106.099} C_VEL
LIN {X 0,Y 237.005,Z 395.355,A -85,B 0,C 180,E1 -21108.33,E2 -21108.33} C_VEL
LIN {X 0,Y 239.058,Z 405.774,A -85,B 0,C 180,E1 -21110.508,E2 -21110.508} C_VEL
LIN {X 0,Y 239.347,Z 408.62,A -85,B 0,C 180,E1 -21111.088,E2 -21111.088} C_VEL
LIN {X 0,Y 235.768,Z 421.132,A -85,B 0,C 180,E1 -21112.869,E2 -21112.869} C_VEL
LIN {X 0,Y 231.788,Z 432.577,A -85,B 0,C 180,E1 -21114.823,E2 -21114.823} C_VEL
LIN {X 0,Y 227.644,Z 444.032,A -85,B 0,C 180,E1 -21117.297,E2 -21117.297} C_VEL
LIN {X 0,Y 223.766,Z 453.659,A -85,B 0,C 180,E1 -21119.832,E2 -21119.832} C_VEL
LIN {X 0,Y 219.596,Z 463.064,A -85,B 0,C 180,E1 -21122.866,E2 -21122.866} C_VEL
LIN {X 0,Y 215.667,Z 471.53,A -85,B 0,C 180,E1 -21126.303,E2 -21126.303} C_VEL
LIN {X 0,Y 212.577,Z 478.128,A -85,B 0,C 180,E1 -21129.687,E2 -21129.687} C_VEL
LIN {X 0,Y 209.917,Z 483.858,A -85,B 0,C 180,E1 -21133.466,E2 -21133.466} C_VEL
LIN {X 0,Y 208.323,Z 487.238,A -85,B 0,C 180,E1 -21136.34,E2 -21136.34} C_VEL
LIN {X 0,Y 206.82,Z 490.668,A -85,B 0,C 180,E1 -21140.217,E2 -21140.217} C_VEL
LIN {X 0,Y 205.896,Z 492.922,A -85,B 0,C 180,E1 -21144.122,E2 -21144.122} C_VEL
LIN {X 0,Y 205.799,Z 493.613,A -85,B 0,C 180,E1 -21146.083,E2 -21146.083} C_VEL
LIN {X 0,Y 205.523,Z 494.203,A -85,B 0,C 180,E1 -21150,E2 -21150} C_VEL
LIN {X 0,Y 205.775,Z 493.645,A -85,B 0,C 180,E1 -21153.916,E2 -21153.916} C_VEL
LIN {X 0,Y 206.237,Z 492.013,A -85,B 0,C 180,E1 -21157.834,E2 -21157.834} C_VEL
LIN {X 0,Y 207.486,Z 489.225,A -85,B 0,C 180,E1 -21161.726,E2 -21161.726} C_VEL
LIN {X 0,Y 209.311,Z 485.229,A -85,B 0,C 180,E1 -21165.581,E2 -21165.581} C_VEL
LIN {X 0,Y 211.802,Z 479.905,A -85,B 0,C 180,E1 -21169.379,E2 -21169.379} C_VEL
LIN {X 0,Y 215.034,Z 473.097,A -85,B 0,C 180,E1 -21173.091,E2 -21173.091} C_VEL
LIN {X 0,Y 218.404,Z 465.792,A -85,B 0,C 180,E1 -21176.261,E2 -21176.261} C_VEL
LIN {X 0,Y 222.398,Z 456.957,A -85,B 0,C 180,E1 -21179.328,E2 -21179.328} C_VEL
LIN {X 0,Y 226.268,Z 447.901,A -85,B 0,C 180,E1 -21181.872,E2 -21181.872} C_VEL
LIN {X 0,Y 229.994,Z 437.873,A -85,B 0,C 180,E1 -21184.237,E2 -21184.237} C_VEL
LIN {X 0,Y 234.06,Z 426.599,A -85,B 0,C 180,E1 -21186.372,E2 -21186.372} C_VEL
LIN {X 0,Y 237.991,Z 413.958,A -85,B 0,C 180,E1 -21188.326,E2 -21188.326} C_VEL
LIN {X 0,Y 239.352,Z 408.996,A -85,B 0,C 180,E1 -21188.992,E2 -21188.992} C_VEL
LIN {X 0,Y 239.016,Z 404.912,A -85,B 0,C 180,E1 -21189.809,E2 -21189.809} C_VEL
LIN {X 0,Y 236.758,Z 394.002,A -85,B 0,C 180,E1 -21192.088,E2 -21192.088} C_VEL
LIN {X 0,Y 233.611,Z 383.016,A -85,B 0,C 180,E1 -21194.397,E2 -21194.397} C_VEL
LIN {X 0,Y 229.254,Z 371.925,A -85,B 0,C 180,E1 -21196.857,E2 -21196.857} C_VEL
LIN {X 0,Y 223.604,Z 361.404,A -85,B 0,C 180,E1 -21199.515,E2 -21199.515} C_VEL
LIN {X 0,Y 220.255,Z 356.287,A -85,B 0,C 180,E1 -21201.001,E2 -21201.001} C_VEL
LIN {X 0,Y 217.87,Z 352.765,A -85,B 0,C 180,E1 -21202.038,E2 -21202.038} C_VEL
LIN {X 0,Y 215.166,Z 348.921,A -85,B 0,C 180,E1 -21203.245,E2 -21203.245} C_VEL
LIN {X 0,Y 212.063,Z 345.145,A -85,B 0,C 180,E1 -21204.624,E2 -21204.624} C_VEL
LIN {X 0,Y 211.186,Z 343.404,A -85,B 0,C 180,E1 -21205.111,E2 -21205.111} C_VEL
LIN {X 0,Y 210.823,Z 341.469,A -85,B 0,C 180,E1 -21207.766,E2 -21207.766} C_VEL
LIN {X 0,Y 210.263,Z 338.681,A -85,B 0,C 180,E1 -21212.099,E2 -21212.099} C_VEL
LIN {X 0,Y 209.797,Z 336.271,A -85,B 0,C 180,E1 -21216.297,E2 -21216.297} C_VEL
LIN {X 0,Y 209.412,Z 334.37,A -85,B 0,C 180,E1 -21220.39,E2 -21220.39} C_VEL
LIN {X 0,Y 209.071,Z 332.646,A -85,B 0,C 180,E1 -21224.4,E2 -21224.4} C_VEL
LIN {X 0,Y 208.877,Z 330.873,A -85,B 0,C 180,E1 -21230.315,E2 -21230.315} C_VEL
LIN {X 0,Y 208.883,Z 330.523,A -85,B 0,C 180,E1 -21232.265,E2 -21232.265} C_VEL
LIN {X 0,Y 208.775,Z 329.703,A -85,B 0,C 180,E1 -21238.071,E2 -21238.071} C_VEL
LIN {X 0,Y 208.915,Z 329.669,A -85,B 0,C 180,E1 -21240,E2 -21240} C_VEL
LIN {X 0,Y 208.937,Z 329.921,A -85,B 0,C 180,E1 -21241.927,E2 -21241.927} C_VEL
LIN {X 0,Y 209.242,Z 331.123,A -85,B 0,C 180,E1 -21247.721,E2 -21247.721} C_VEL
LIN {X 0,Y 209.49,Z 331.718,A -85,B 0,C 180,E1 -21249.656,E2 -21249.656} C_VEL
LIN {X 0,Y 210.404,Z 334.577,A -85,B 0,C 180,E1 -21255.499,E2 -21255.499} C_VEL
LIN {X 0,Y 211.37,Z 337.353,A -85,B 0,C 180,E1 -21259.42,E2 -21259.42} C_VEL
LIN {X 0,Y 213.24,Z 341.788,A -85,B 0,C 180,E1 -21264.329,E2 -21264.329} C_VEL
LIN {X 0,Y 214.929,Z 345.813,A -85,B 0,C 180,E1 -21268.009,E2 -21268.009} C_VEL
LIN {X 0,Y 215.855,Z 350.875,A -85,B 0,C 180,E1 -21271.395,E2 -21271.395} C_VEL
LIN {X 0,Y 217.642,Z 360.083,A -85,B 0,C 180,E1 -21276.682,E2 -21276.682} C_VEL
LIN {X 0,Y 218.064,Z 361.881,A -85,B 0,C 180,E1 -21277.541,E2 -21277.541} C_VEL
LIN {X 0,Y 220.958,Z 367.114,A -85,B 0,C 180,E1 -21278.755,E2 -21278.755} C_VEL
LIN {X 0,Y 225.171,Z 374.881,A -85,B 0,C 180,E1 -21280.438,E2 -21280.438} C_VEL
LIN {X 0,Y 230.139,Z 384.714,A -85,B 0,C 180,E1 -21282.431,E2 -21282.431} C_VEL
LIN {X 0,Y 233.999,Z 393.279,A -85,B 0,C 180,E1 -21284.065,E2 -21284.065} C_VEL
LIN {X 0,Y 235.176,Z 406.538,A -85,B 0,C 180,E1 -21285.595,E2 -21285.595} C_VEL
LIN {X 0,Y 235.344,Z 417.597,A -85,B 0,C 180,E1 -21286.946,E2 -21286.946} C_VEL
LIN {X 0,Y 234.621,Z 431.483,A -85,B 0,C 180,E1 -21288.776,E2 -21288.776} C_VEL
LIN {X 0,Y 233.289,Z 444.039,A -85,B 0,C 180,E1 -21290.659,E2 -21290.659} C_VEL
LIN {X 0,Y 232.459,Z 447.399,A -85,B 0,C 180,E1 -21291.145,E2 -21291.145} C_VEL
LIN {X 0,Y 231.052,Z 450.715,A -85,B 0,C 180,E1 -21291.552,E2 -21291.552} C_VEL
LIN {X 0,Y 227.21,Z 457.081,A -85,B 0,C 180,E1 -21292.245,E2 -21292.245} C_VEL
LIN {X 0,Y 222.001,Z 464.798,A -85,B 0,C 180,E1 -21293.202,E2 -21293.202} C_VEL
LIN {X 0,Y 219.634,Z 469.306,A -85,B 0,C 180,E1 -21294.011,E2 -21294.011} C_VEL
LIN {X 0,Y 215.391,Z 479.399,A -85,B 0,C 180,E1 -21296.311,E2 -21296.311} C_VEL
LIN {X 0,Y 211.355,Z 488.847,A -85,B 0,C 180,E1 -21298.976,E2 -21298.976} C_VEL
LIN {X 0,Y 207.325,Z 498.14,A -85,B 0,C 180,E1 -21302.219,E2 -21302.219} C_VEL
LIN {X 0,Y 204.001,Z 505.883,A -85,B 0,C 180,E1 -21305.581,E2 -21305.581} C_VEL
LIN {X 0,Y 201.049,Z 513.147,A -85,B 0,C 180,E1 -21309.54,E2 -21309.54} C_VEL
LIN {X 0,Y 199.073,Z 518.897,A -85,B 0,C 180,E1 -21313.595,E2 -21313.595} C_VEL
LIN {X 0,Y 198.005,Z 523.276,A -85,B 0,C 180,E1 -21317.704,E2 -21317.704} C_VEL
LIN {X 0,Y 197.751,Z 526.388,A -85,B 0,C 180,E1 -21321.828,E2 -21321.828} C_VEL
LIN {X 0,Y 197.949,Z 527.494,A -85,B 0,C 180,E1 -21323.886,E2 -21323.886} C_VEL
LIN {X 0,Y 198.209,Z 528.767,A -85,B 0,C 180,E1 -21327.968,E2 -21327.968} C_VEL
LIN {X 0,Y 198.499,Z 528.954,A -85,B 0,C 180,E1 -21330,E2 -21330} C_VEL
LIN {X 0,Y 198.061,Z 528.274,A -85,B 0,C 180,E1 -21334.07,E2 -21334.07} C_VEL
LIN {X 0,Y 197.948,Z 527.436,A -85,B 0,C 180,E1 -21336.218,E2 -21336.218} C_VEL
LIN {X 0,Y 197.821,Z 524.958,A -85,B 0,C 180,E1 -21340.233,E2 -21340.233} C_VEL
LIN {X 0,Y 198.456,Z 521.199,A -85,B 0,C 180,E1 -21344.353,E2 -21344.353} C_VEL
LIN {X 0,Y 199.982,Z 516.131,A -85,B 0,C 180,E1 -21348.439,E2 -21348.439} C_VEL
LIN {X 0,Y 202.367,Z 509.625,A -85,B 0,C 180,E1 -21352.459,E2 -21352.459} C_VEL
LIN {X 0,Y 205.866,Z 501.515,A -85,B 0,C 180,E1 -21356.347,E2 -21356.347} C_VEL
LIN {X 0,Y 209.048,Z 494.468,A -85,B 0,C 180,E1 -21359.204,E2 -21359.204} C_VEL
LIN {X 0,Y 215.981,Z 487.84,A -85,B 0,C 180,E1 -21363.586,E2 -21363.586} C_VEL
LIN {X 0,Y 222.738,Z 481.486,A -85,B 0,C 180,E1 -21366.835,E2 -21366.835} C_VEL
LIN {X 0,Y 230.628,Z 474.233,A -85,B 0,C 180,E1 -21369.788,E2 -21369.788} C_VEL
LIN {X 0,Y 240.607,Z 464.831,A -85,B 0,C 180,E1 -21372.776,E2 -21372.776} C_VEL
LIN {X 0,Y 245.561,Z 459.938,A -85,B 0,C 180,E1 -21374.129,E2 -21374.129} C_VEL
LIN {X 0,Y 252.684,Z 452.172,A -85,B 0,C 180,E1 -21376.316,E2 -21376.316} C_VEL
LIN {X 0,Y 256.52,Z 447.644,A -85,B 0,C 180,E1 -21377.709,E2 -21377.709} C_VEL
LIN {X 0,Y 257.467,Z 445.686,A -85,B 0,C 180,E1 -21379.071,E2 -21379.071} C_VEL
LIN {X 0,Y 257.351,Z 444.542,A -85,B 0,C 180,E1 -21381.09,E2 -21381.09} C_VEL
LIN {X 0,Y 256.455,Z 444.511,A -85,B 0,C 180,E1 -21383.446,E2 -21383.446} C_VEL
LIN {X 0,Y 254.305,Z 446.1,A -85,B 0,C 180,E1 -21384.524,E2 -21384.524} C_VEL
LIN {X 0,Y 245.38,Z 452.288,A -85,B 0,C 180,E1 -21387.031,E2 -21387.031} C_VEL
LIN {X 0,Y 237.168,Z 457.176,A -85,B 0,C 180,E1 -21389.751,E2 -21389.751} C_VEL
LIN {X 0,Y 229.612,Z 460.906,A -85,B 0,C 180,E1 -21392.67,E2 -21392.67} C_VEL
LIN {X 0,Y 222.84,Z 463.454,A -85,B 0,C 180,E1 -21395.795,E2 -21395.795} C_VEL
LIN {X 0,Y 216.918,Z 464.824,A -85,B 0,C 180,E1 -21399.121,E2 -21399.121} C_VEL
LIN {X 0,Y 211.823,Z 465.047,A -85,B 0,C 180,E1 -21402.626,E2 -21402.626} C_VEL
LIN {X 0,Y 207.607,Z 464.054,A -85,B 0,C 180,E1 -21406.293,E2 -21406.293} C_VEL
LIN {X 0,Y 204.408,Z 461.77,A -85,B 0,C 180,E1 -21410.101,E2 -21410.101} C_VEL
LIN {X 0,Y 202.184,Z 458.172,A -85,B 0,C 180,E1 -21414.014,E2 -21414.014} C_VEL
LIN {X 0,Y 200.59,Z 453.149,A -85,B 0,C 180,E1 -21417.992,E2 -21417.992} C_VEL
LIN {X 0,Y 199.836,Z 448.411,A -85,B 0,C 180,E1 -21421.008,E2 -21421.008} C_VEL
LIN {X 0,Y 199.529,Z 441.634,A -85,B 0,C 180,E1 -21424.546,E2 -21424.546} C_VEL
LIN {X 0,Y 200.145,Z 432.103,A -85,B 0,C 180,E1 -21428.583,E2 -21428.583} C_VEL
LIN {X 0,Y 201.009,Z 421.889,A -85,B 0,C 180,E1 -21432.11,E2 -21432.11} C_VEL
LIN {X 0,Y 202.103,Z 411.347,A -85,B 0,C 180,E1 -21435.118,E2 -21435.118} C_VEL
LIN {X 0,Y 203.485,Z 398.719,A -85,B 0,C 180,E1 -21438.11,E2 -21438.11} C_VEL
LIN {X 0,Y 205.342,Z 384.839,A -85,B 0,C 180,E1 -21440.799,E2 -21440.799} C_VEL
LIN {X 0,Y 206.94,Z 370.435,A -85,B 0,C 180,E1 -21443.068,E2 -21443.068} C_VEL
LIN {X 0,Y 206.997,Z 367.099,A -85,B 0,C 180,E1 -21443.549,E2 -21443.549} C_VEL
LIN {X 0,Y 203.603,Z 351.694,A -85,B 0,C 180,E1 -21445.652,E2 -21445.652} C_VEL
LIN {X 0,Y 201.464,Z 341.965,A -85,B 0,C 180,E1 -21446.84,E2 -21446.84} C_VEL
LIN {X 0,Y 202.666,Z 342.802,A -85,B 0,C 180,E1 -21449.045,E2 -21449.045} C_VEL
LIN {X 0,Y 203.72,Z 344.466,A -85,B 0,C 180,E1 -21452.034,E2 -21452.034} C_VEL
LIN {X 0,Y 206.01,Z 347.722,A -85,B 0,C 180,E1 -21453.263,E2 -21453.263} C_VEL
LIN {X 0,Y 208.498,Z 350.071,A -85,B 0,C 180,E1 -21454.458,E2 -21454.458} C_VEL
LIN {X 0,Y 211.149,Z 353.719,A -85,B 0,C 180,E1 -21455.772,E2 -21455.772} C_VEL
LIN {X 0,Y 212.597,Z 355.702,A -85,B 0,C 180,E1 -21456.466,E2 -21456.466} C_VEL
LIN {X 0,Y 215.904,Z 360.488,A -85,B 0,C 180,E1 -21458.057,E2 -21458.057} C_VEL
LIN {X 0,Y 218.771,Z 365.081,A -85,B 0,C 180,E1 -21459.441,E2 -21459.441} C_VEL
LIN {X 0,Y 223.079,Z 372.985,A -85,B 0,C 180,E1 -21461.641,E2 -21461.641} C_VEL
LIN {X 0,Y 225.878,Z 379.182,A -85,B 0,C 180,E1 -21463.197,E2 -21463.197} C_VEL
LIN {X 0,Y 229.499,Z 390.269,A -85,B 0,C 180,E1 -21465.711,E2 -21465.711} C_VEL
LIN {X 0,Y 231.927,Z 400.385,A -85,B 0,C 180,E1 -21467.939,E2 -21467.939} C_VEL
LIN {X 0,Y 233.533,Z 410.492,A -85,B 0,C 180,E1 -21470.16,E2 -21470.16} C_VEL
LIN {X 0,Y 229.756,Z 422.988,A -85,B 0,C 180,E1 -21472.004,E2 -21472.004} C_VEL
LIN {X 0,Y 226.043,Z 433.179,A -85,B 0,C 180,E1 -21473.79,E2 -21473.79} C_VEL
LIN {X 0,Y 221.727,Z 444.636,A -85,B 0,C 180,E1 -21476.31,E2 -21476.31} C_VEL
LIN {X 0,Y 217.692,Z 454.263,A -85,B 0,C 180,E1 -21478.899,E2 -21478.899} C_VEL
LIN {X 0,Y 213.316,Z 463.672,A -85,B 0,C 180,E1 -21481.998,E2 -21481.998} C_VEL
LIN {X 0,Y 209.76,Z 471.029,A -85,B 0,C 180,E1 -21484.993,E2 -21484.993} C_VEL
LIN {X 0,Y 206.744,Z 477.066,A -85,B 0,C 180,E1 -21488.041,E2 -21488.041} C_VEL
LIN {X 0,Y 203.789,Z 483.149,A -85,B 0,C 180,E1 -21491.917,E2 -21491.917} C_VEL
LIN {X 0,Y 201.451,Z 487.848,A -85,B 0,C 180,E1 -21495.864,E2 -21495.864} C_VEL
LIN {X 0,Y 199.802,Z 491.386,A -85,B 0,C 180,E1 -21500.03,E2 -21500.03} C_VEL
LIN {X 0,Y 198.849,Z 493.531,A -85,B 0,C 180,E1 -21503.913,E2 -21503.913} C_VEL
LIN {X 0,Y 198.742,Z 494.222,A -85,B 0,C 180,E1 -21505.944,E2 -21505.944} C_VEL
LIN {X 0,Y 198.478,Z 494.809,A -85,B 0,C 180,E1 -21510,E2 -21510} C_VEL
LIN {X 0,Y 198.72,Z 494.253,A -85,B 0,C 180,E1 -21514.056,E2 -21514.056} C_VEL
LIN {X 0,Y 199.24,Z 492.62,A -85,B 0,C 180,E1 -21518.111,E2 -21518.111} C_VEL
LIN {X 0,Y 200.55,Z 489.834,A -85,B 0,C 180,E1 -21522.137,E2 -21522.137} C_VEL
LIN {X 0,Y 202.478,Z 485.838,A -85,B 0,C 180,E1 -21526.121,E2 -21526.121} C_VEL
LIN {X 0,Y 205.112,Z 480.513,A -85,B 0,C 180,E1 -21530.037,E2 -21530.037} C_VEL
LIN {X 0,Y 208.508,Z 473.705,A -85,B 0,C 180,E1 -21533.858,E2 -21533.858} C_VEL
LIN {X 0,Y 212.075,Z 466.396,A -85,B 0,C 180,E1 -21537.107,E2 -21537.107} C_VEL
LIN {X 0,Y 216.244,Z 457.56,A -85,B 0,C 180,E1 -21540.248,E2 -21540.248} C_VEL
LIN {X 0,Y 220.28,Z 448.503,A -85,B 0,C 180,E1 -21542.846,E2 -21542.846} C_VEL
LIN {X 0,Y 224.497,Z 437.665,A -85,B 0,C 180,E1 -21545.43,E2 -21545.43} C_VEL
LIN {X 0,Y 228.804,Z 426.051,A -85,B 0,C 180,E1 -21547.624,E2 -21547.624} C_VEL
LIN {X 0,Y 232.821,Z 413.357,A -85,B 0,C 180,E1 -21549.579,E2 -21549.579} C_VEL
LIN {X 0,Y 233.568,Z 410.845,A -85,B 0,C 180,E1 -21549.919,E2 -21549.919} C_VEL
LIN {X 0,Y 232.463,Z 402.662,A -85,B 0,C 180,E1 -21551.691,E2 -21551.691} C_VEL
LIN {X 0,Y 229.995,Z 391.797,A -85,B 0,C 180,E1 -21554.104,E2 -21554.104} C_VEL
LIN {X 0,Y 226.766,Z 381.606,A -85,B 0,C 180,E1 -21556.403,E2 -21556.403} C_VEL
LIN {X 0,Y 223.42,Z 373.67,A -85,B 0,C 180,E1 -21558.353,E2 -21558.353} C_VEL
LIN {X 0,Y 218.843,Z 365.186,A -85,B 0,C 180,E1 -21560.709,E2 -21560.709} C_VEL
LIN {X 0,Y 214.39,Z 358.14,A -85,B 0,C 180,E1 -21562.887,E2 -21562.887} C_VEL
LIN {X 0,Y 211.278,Z 353.753,A -85,B 0,C 180,E1 -21564.376,E2 -21564.376} C_VEL
LIN {X 0,Y 208.761,Z 350.211,A -85,B 0,C 180,E1 -21565.633,E2 -21565.633} C_VEL
LIN {X 0,Y 207.477,Z 348.792,A -85,B 0,C 180,E1 -21566.255,E2 -21566.255} C_VEL
LIN {X 0,Y 204.987,Z 345.641,A -85,B 0,C 180,E1 -21567.535,E2 -21567.535} C_VEL
LIN {X 0,Y 204.341,Z 344.315,A -85,B 0,C 180,E1 -21567.93,E2 -21567.93} C_VEL
LIN {X 0,Y 203.935,Z 342.29,A -85,B 0,C 180,E1 -21571.153,E2 -21571.153} C_VEL
LIN {X 0,Y 203.467,Z 339.814,A -85,B 0,C 180,E1 -21575.512,E2 -21575.512} C_VEL
LIN {X 0,Y 203.11,Z 337.8,A -85,B 0,C 180,E1 -21579.756,E2 -21579.756} C_VEL
LIN {X 0,Y 202.803,Z 336.165,A -85,B 0,C 180,E1 -21583.905,E2 -21583.905} C_VEL
LIN {X 0,Y 202.672,Z 335.028,A -85,B 0,C 180,E1 -21587.991,E2 -21587.991} C_VEL
LIN {X 0,Y 202.682,Z 334.001,A -85,B 0,C 180,E1 -21592.027,E2 -21592.027} C_VEL
LIN {X 0,Y 202.737,Z 333.465,A -85,B 0,C 180,E1 -21598.013,E2 -21598.013} C_VEL
LIN {X 0,Y 202.885,Z 333.423,A -85,B 0,C 180,E1 -21600,E2 -21600} C_VEL
LIN {X 0,Y 202.823,Z 334.149,A -85,B 0,C 180,E1 -21603.974,E2 -21603.974} C_VEL
LIN {X 0,Y 203.361,Z 335.11,A -85,B 0,C 180,E1 -21607.946,E2 -21607.946} C_VEL
LIN {X 0,Y 203.756,Z 336.78,A -85,B 0,C 180,E1 -21611.944,E2 -21611.944} C_VEL
LIN {X 0,Y 204.755,Z 339.056,A -85,B 0,C 180,E1 -21616.041,E2 -21616.041} C_VEL
LIN {X 0,Y 205.759,Z 341.963,A -85,B 0,C 180,E1 -21619.972,E2 -21619.972} C_VEL
LIN {X 0,Y 207.27,Z 345.529,A -85,B 0,C 180,E1 -21624.009,E2 -21624.009} C_VEL
LIN {X 0,Y 208.718,Z 348.739,A -85,B 0,C 180,E1 -21627.037,E2 -21627.037} C_VEL
LIN {X 0,Y 209.643,Z 353.054,A -85,B 0,C 180,E1 -21630.189,E2 -21630.189} C_VEL
LIN {X 0,Y 211.05,Z 361.09,A -85,B 0,C 180,E1 -21634.987,E2 -21634.987} C_VEL
LIN {X 0,Y 214.207,Z 366.5,A -85,B 0,C 180,E1 -21636.452,E2 -21636.452} C_VEL
LIN {X 0,Y 220.846,Z 378.79,A -85,B 0,C 180,E1 -21639.372,E2 -21639.372} C_VEL
LIN {X 0,Y 225.958,Z 389.637,A -85,B 0,C 180,E1 -21641.667,E2 -21641.667} C_VEL
LIN {X 0,Y 229.015,Z 396.793,A -85,B 0,C 180,E1 -21643.121,E2 -21643.121} C_VEL
LIN {X 0,Y 229.805,Z 409.566,A -85,B 0,C 180,E1 -21644.7,E2 -21644.7} C_VEL
LIN {X 0,Y 229.713,Z 421.038,A -85,B 0,C 180,E1 -21646.174,E2 -21646.174} C_VEL
LIN {X 0,Y 228.701,Z 433.937,A -85,B 0,C 180,E1 -21647.974,E2 -21647.974} C_VEL
LIN {X 0,Y 226.859,Z 448.28,A -85,B 0,C 180,E1 -21650.287,E2 -21650.287} C_VEL
LIN {X 0,Y 225.949,Z 452.237,A -85,B 0,C 180,E1 -21650.962,E2 -21650.962} C_VEL
LIN {X 0,Y 221.279,Z 465.088,A -85,B 0,C 180,E1 -21653.167,E2 -21653.167} C_VEL
LIN {X 0,Y 219.634,Z 469.306,A -85,B 0,C 180,E1 -21654.011,E2 -21654.011} C_VEL
LIN {X 0,Y 217.305,Z 473.684,A -85,B 0,C 180,E1 -21654.865,E2 -21654.865} C_VEL
LIN {X 0,Y 211.887,Z 480.46,A -85,B 0,C 180,E1 -21656.151,E2 -21656.151} C_VEL
LIN {X 0,Y 206.475,Z 486.849,A -85,B 0,C 180,E1 -21657.594,E2 -21657.594} C_VEL
LIN {X 0,Y 204.163,Z 490.53,A -85,B 0,C 180,E1 -21658.702,E2 -21658.702} C_VEL
LIN {X 0,Y 199.919,Z 499.866,A -85,B 0,C 180,E1 -21662.239,E2 -21662.239} C_VEL
LIN {X 0,Y 196.56,Z 507.239,A -85,B 0,C 180,E1 -21665.721,E2 -21665.721} C_VEL
LIN {X 0,Y 193.692,Z 514.11,A -85,B 0,C 180,E1 -21669.837,E2 -21669.837} C_VEL
LIN {X 0,Y 191.777,Z 519.518,A -85,B 0,C 180,E1 -21674.047,E2 -21674.047} C_VEL
LIN {X 0,Y 190.984,Z 522.659,A -85,B 0,C 180,E1 -21677.245,E2 -21677.245} C_VEL
LIN {X 0,Y 190.672,Z 525.773,A -85,B 0,C 180,E1 -21681.522,E2 -21681.522} C_VEL
LIN {X 0,Y 190.868,Z 526.944,A -85,B 0,C 180,E1 -21683.811,E2 -21683.811} C_VEL
LIN {X 0,Y 191.116,Z 528.157,A -85,B 0,C 180,E1 -21687.893,E2 -21687.893} C_VEL
LIN {X 0,Y 191.441,Z 528.347,A -85,B 0,C 180,E1 -21690,E2 -21690} C_VEL
LIN {X 0,Y 190.983,Z 527.663,A -85,B 0,C 180,E1 -21694.221,E2 -21694.221} C_VEL
LIN {X 0,Y 190.842,Z 526.864,A -85,B 0,C 180,E1 -21696.343,E2 -21696.343} C_VEL
LIN {X 0,Y 190.752,Z 524.34,A -85,B 0,C 180,E1 -21700.616,E2 -21700.616} C_VEL
LIN {X 0,Y 191.492,Z 520.58,A -85,B 0,C 180,E1 -21704.887,E2 -21704.887} C_VEL
LIN {X 0,Y 193.14,Z 515.509,A -85,B 0,C 180,E1 -21709.117,E2 -21709.117} C_VEL
LIN {X 0,Y 195.746,Z 509.007,A -85,B 0,C 180,E1 -21713.263,E2 -21713.263} C_VEL
LIN {X 0,Y 199.435,Z 500.897,A -85,B 0,C 180,E1 -21717.266,E2 -21717.266} C_VEL
LIN {X 0,Y 202.345,Z 494.564,A -85,B 0,C 180,E1 -21719.845,E2 -21719.845} C_VEL
LIN {X 0,Y 208.463,Z 489.301,A -85,B 0,C 180,E1 -21723.799,E2 -21723.799} C_VEL
LIN {X 0,Y 217.116,Z 482.028,A -85,B 0,C 180,E1 -21727.955,E2 -21727.955} C_VEL
LIN {X 0,Y 227.504,Z 473.356,A -85,B 0,C 180,E1 -21731.62,E2 -21731.62} C_VEL
LIN {X 0,Y 237.995,Z 464.26,A -85,B 0,C 180,E1 -21734.535,E2 -21734.535} C_VEL
LIN {X 0,Y 247.036,Z 455.526,A -85,B 0,C 180,E1 -21737.102,E2 -21737.102} C_VEL
LIN {X 0,Y 250.143,Z 452.332,A -85,B 0,C 180,E1 -21738.12,E2 -21738.12} C_VEL
LIN {X 0,Y 251.574,Z 450.526,A -85,B 0,C 180,E1 -21738.963,E2 -21738.963} C_VEL
LIN {X 0,Y 251.88,Z 449.517,A -85,B 0,C 180,E1 -21740.078,E2 -21740.078} C_VEL
LIN {X 0,Y 251.462,Z 448.856,A -85,B 0,C 180,E1 -21742.058,E2 -21742.058} C_VEL
LIN {X 0,Y 250.995,Z 448.869,A -85,B 0,C 180,E1 -21742.986,E2 -21742.986} C_VEL
LIN {X 0,Y 249.187,Z 449.988,A -85,B 0,C 180,E1 -21743.681,E2 -21743.681} C_VEL
LIN {X 0,Y 239.991,Z 455.659,A -85,B 0,C 180,E1 -21746.193,E2 -21746.193} C_VEL
LIN {X 0,Y 231.506,Z 460.098,A -85,B 0,C 180,E1 -21748.93,E2 -21748.93} C_VEL
LIN {X 0,Y 223.706,Z 463.414,A -85,B 0,C 180,E1 -21751.885,E2 -21751.885} C_VEL
LIN {X 0,Y 216.665,Z 465.59,A -85,B 0,C 180,E1 -21755.059,E2 -21755.059} C_VEL
LIN {X 0,Y 210.503,Z 466.605,A -85,B 0,C 180,E1 -21758.454,E2 -21758.454} C_VEL
LIN {X 0,Y 205.194,Z 466.466,A -85,B 0,C 180,E1 -21762.046,E2 -21762.046} C_VEL
LIN {X 0,Y 200.818,Z 465.118,A -85,B 0,C 180,E1 -21765.82,E2 -21765.82} C_VEL
LIN {X 0,Y 197.455,Z 462.495,A -85,B 0,C 180,E1 -21769.749,E2 -21769.749} C_VEL
LIN {X 0,Y 195.132,Z 458.565,A -85,B 0,C 180,E1 -21773.797,E2 -21773.797} C_VEL
LIN {X 0,Y 193.482,Z 453.262,A -85,B 0,C 180,E1 -21777.919,E2 -21777.919} C_VEL
LIN {X 0,Y 192.731,Z 448.259,A -85,B 0,C 180,E1 -21781.045,E2 -21781.045} C_VEL
LIN {X 0,Y 192.475,Z 440.12,A -85,B 0,C 180,E1 -21785.238,E2 -21785.238} C_VEL
LIN {X 0,Y 193.132,Z 431.229,A -85,B 0,C 180,E1 -21788.933,E2 -21788.933} C_VEL
LIN {X 0,Y 194.053,Z 420.713,A -85,B 0,C 180,E1 -21792.551,E2 -21792.551} C_VEL
LIN {X 0,Y 195.204,Z 409.837,A -85,B 0,C 180,E1 -21795.666,E2 -21795.666} C_VEL
LIN {X 0,Y 196.541,Z 397.947,A -85,B 0,C 180,E1 -21798.503,E2 -21798.503} C_VEL
LIN {X 0,Y 198.275,Z 385.136,A -85,B 0,C 180,E1 -21801.032,E2 -21801.032} C_VEL
LIN {X 0,Y 199.919,Z 370.85,A -85,B 0,C 180,E1 -21803.337,E2 -21803.337} C_VEL
LIN {X 0,Y 200.078,Z 369.221,A -85,B 0,C 180,E1 -21803.575,E2 -21803.575} C_VEL
LIN {X 0,Y 197.217,Z 355.353,A -85,B 0,C 180,E1 -21805.585,E2 -21805.585} C_VEL
LIN {X 0,Y 194.958,Z 345.214,A -85,B 0,C 180,E1 -21806.901,E2 -21806.901} C_VEL
LIN {X 0,Y 195.787,Z 345.644,A -85,B 0,C 180,E1 -21808.108,E2 -21808.108} C_VEL
LIN {X 0,Y 199.758,Z 349.821,A -85,B 0,C 180,E1 -21810.509,E2 -21810.509} C_VEL
LIN {X 0,Y 201.52,Z 351.215,A -85,B 0,C 180,E1 -21811.465,E2 -21811.465} C_VEL
LIN {X 0,Y 204.409,Z 354.874,A -85,B 0,C 180,E1 -21813.081,E2 -21813.081} C_VEL
LIN {X 0,Y 205.851,Z 356.399,A -85,B 0,C 180,E1 -21813.829,E2 -21813.829} C_VEL
LIN {X 0,Y 209.516,Z 361.642,A -85,B 0,C 180,E1 -21815.798,E2 -21815.798} C_VEL
LIN {X 0,Y 212.641,Z 366.391,A -85,B 0,C 180,E1 -21817.447,E2 -21817.447} C_VEL
LIN {X 0,Y 216.893,Z 373.988,A -85,B 0,C 180,E1 -21819.797,E2 -21819.797} C_VEL
LIN {X 0,Y 220.565,Z 381.93,A -85,B 0,C 180,E1 -21822.001,E2 -21822.001} C_VEL
LIN {X 0,Y 223.901,Z 392.24,A -85,B 0,C 180,E1 -21824.494,E2 -21824.494} C_VEL
LIN {X 0,Y 226.237,Z 402.465,A -85,B 0,C 180,E1 -21826.887,E2 -21826.887} C_VEL
LIN {X 0,Y 227.738,Z 412.35,A -85,B 0,C 180,E1 -21829.176,E2 -21829.176} C_VEL
LIN {X 0,Y 223.794,Z 424.845,A -85,B 0,C 180,E1 -21831.091,E2 -21831.091} C_VEL
LIN {X 0,Y 219.61,Z 435.893,A -85,B 0,C 180,E1 -21833.136,E2 -21833.136} C_VEL
LIN {X 0,Y 215.146,Z 446.975,A -85,B 0,C 180,E1 -21835.702,E2 -21835.702} C_VEL
LIN {X 0,Y 210.927,Z 456.319,A -85,B 0,C 180,E1 -21838.346,E2 -21838.346} C_VEL
LIN {X 0,Y 206.491,Z 465.475,A -85,B 0,C 180,E1 -21841.543,E2 -21841.543} C_VEL
LIN {X 0,Y 202.673,Z 472.936,A -85,B 0,C 180,E1 -21844.786,E2 -21844.786} C_VEL
LIN {X 0,Y 199.319,Z 479.349,A -85,B 0,C 180,E1 -21848.27,E2 -21848.27} C_VEL
LIN {X 0,Y 196.352,Z 485.079,A -85,B 0,C 180,E1 -21852.287,E2 -21852.287} C_VEL
LIN {X 0,Y 194.58,Z 488.458,A -85,B 0,C 180,E1 -21855.354,E2 -21855.354} C_VEL
LIN {X 0,Y 192.782,Z 492.108,A -85,B 0,C 180,E1 -21859.836,E2 -21859.836} C_VEL
LIN {X 0,Y 191.808,Z 494.141,A -85,B 0,C 180,E1 -21863.689,E2 -21863.689} C_VEL
LIN {X 0,Y 191.689,Z 494.83,A -85,B 0,C 180,E1 -21865.794,E2 -21865.794} C_VEL
LIN {X 0,Y 191.413,Z 495.416,A -85,B 0,C 180,E1 -21870,E2 -21870} C_VEL
LIN {X 0,Y 191.651,Z 494.863,A -85,B 0,C 180,E1 -21874.205,E2 -21874.205} C_VEL
LIN {X 0,Y 192.25,Z 493.227,A -85,B 0,C 180,E1 -21878.408,E2 -21878.408} C_VEL
LIN {X 0,Y 193.642,Z 490.441,A -85,B 0,C 180,E1 -21882.577,E2 -21882.577} C_VEL
LIN {X 0,Y 195.672,Z 486.446,A -85,B 0,C 180,E1 -21886.698,E2 -21886.698} C_VEL
LIN {X 0,Y 198.452,Z 481.122,A -85,B 0,C 180,E1 -21890.74,E2 -21890.74} C_VEL
LIN {X 0,Y 202.042,Z 474.311,A -85,B 0,C 180,E1 -21894.671,E2 -21894.671} C_VEL
LIN {X 0,Y 205.807,Z 466.999,A -85,B 0,C 180,E1 -21898.004,E2 -21898.004} C_VEL
LIN {X 0,Y 210.164,Z 458.162,A -85,B 0,C 180,E1 -21901.22,E2 -21901.22} C_VEL
LIN {X 0,Y 214.343,Z 449.105,A -85,B 0,C 180,E1 -21903.876,E2 -21903.876} C_VEL
LIN {X 0,Y 218.79,Z 438.218,A -85,B 0,C 180,E1 -21906.514,E2 -21906.514} C_VEL
LIN {X 0,Y 223.253,Z 426.643,A -85,B 0,C 180,E1 -21908.731,E2 -21908.731} C_VEL
LIN {X 0,Y 227.426,Z 413.92,A -85,B 0,C 180,E1 -21910.718,E2 -21910.718} C_VEL
LIN {X 0,Y 227.807,Z 412.702,A -85,B 0,C 180,E1 -21910.891,E2 -21910.891} C_VEL
LIN {X 0,Y 226.463,Z 403.33,A -85,B 0,C 180,E1 -21913.058,E2 -21913.058} C_VEL
LIN {X 0,Y 224.161,Z 393.033,A -85,B 0,C 180,E1 -21915.475,E2 -21915.475} C_VEL
LIN {X 0,Y 221.518,Z 384.402,A -85,B 0,C 180,E1 -21917.547,E2 -21917.547} C_VEL
LIN {X 0,Y 217.875,Z 375.905,A -85,B 0,C 180,E1 -21919.824,E2 -21919.824} C_VEL
LIN {X 0,Y 213.503,Z 367.84,A -85,B 0,C 180,E1 -21922.271,E2 -21922.271} C_VEL
LIN {X 0,Y 210.504,Z 363.11,A -85,B 0,C 180,E1 -21923.879,E2 -21923.879} C_VEL
LIN {X 0,Y 207.965,Z 359.27,A -85,B 0,C 180,E1 -21925.262,E2 -21925.262} C_VEL
LIN {X 0,Y 205.181,Z 355.233,A -85,B 0,C 180,E1 -21926.767,E2 -21926.767} C_VEL
LIN {X 0,Y 202.486,Z 351.858,A -85,B 0,C 180,E1 -21928.261,E2 -21928.261} C_VEL
LIN {X 0,Y 201.513,Z 350.382,A -85,B 0,C 180,E1 -21928.824,E2 -21928.824} C_VEL
LIN {X 0,Y 198.658,Z 347.428,A -85,B 0,C 180,E1 -21930.457,E2 -21930.457} C_VEL
LIN {X 0,Y 197.52,Z 345.287,A -85,B 0,C 180,E1 -21931.292,E2 -21931.292} C_VEL
LIN {X 0,Y 197.157,Z 343.415,A -85,B 0,C 180,E1 -21934.674,E2 -21934.674} C_VEL
LIN {X 0,Y 196.846,Z 341.329,A -85,B 0,C 180,E1 -21939.082,E2 -21939.082} C_VEL
LIN {X 0,Y 196.551,Z 339.719,A -85,B 0,C 180,E1 -21943.378,E2 -21943.378} C_VEL
LIN {X 0,Y 196.41,Z 338.488,A -85,B 0,C 180,E1 -21947.602,E2 -21947.602} C_VEL
LIN {X 0,Y 196.578,Z 337.705,A -85,B 0,C 180,E1 -21951.778,E2 -21951.778} C_VEL
LIN {X 0,Y 196.675,Z 337.175,A -85,B 0,C 180,E1 -21957.952,E2 -21957.952} C_VEL
LIN {X 0,Y 196.894,Z 337.227,A -85,B 0,C 180,E1 -21960,E2 -21960} C_VEL
LIN {X 0,Y 196.944,Z 338.148,A -85,B 0,C 180,E1 -21964.092,E2 -21964.092} C_VEL
LIN {X 0,Y 197.53,Z 339.234,A -85,B 0,C 180,E1 -21968.182,E2 -21968.182} C_VEL
LIN {X 0,Y 197.985,Z 341.031,A -85,B 0,C 180,E1 -21972.297,E2 -21972.297} C_VEL
LIN {X 0,Y 198.961,Z 343.327,A -85,B 0,C 180,E1 -21976.414,E2 -21976.414} C_VEL
LIN {X 0,Y 200.108,Z 346.504,A -85,B 0,C 180,E1 -21980.561,E2 -21980.561} C_VEL
LIN {X 0,Y 201.917,Z 350.808,A -85,B 0,C 180,E1 -21985.182,E2 -21985.182} C_VEL
LIN {X 0,Y 203.141,Z 353.775,A -85,B 0,C 180,E1 -21987.843,E2 -21987.843} C_VEL
LIN {X 0,Y 204.072,Z 359.909,A -85,B 0,C 180,E1 -21992.044,E2 -21992.044} C_VEL
LIN {X 0,Y 206.916,Z 365.179,A -85,B 0,C 180,E1 -21993.594,E2 -21993.594} C_VEL
LIN {X 0,Y 208.565,Z 367.928,A -85,B 0,C 180,E1 -21994.421,E2 -21994.421} C_VEL
LIN {X 0,Y 211.839,Z 373.714,A -85,B 0,C 180,E1 -21996.023,E2 -21996.023} C_VEL
LIN {X 0,Y 217.037,Z 384.001,A -85,B 0,C 180,E1 -21998.561,E2 -21998.561} C_VEL
LIN {X 0,Y 221.368,Z 393.711,A -85,B 0,C 180,E1 -22000.754,E2 -22000.754} C_VEL
LIN {X 0,Y 223.996,Z 400.414,A -85,B 0,C 180,E1 -22002.182,E2 -22002.182} C_VEL
LIN {X 0,Y 224.494,Z 412.347,A -85,B 0,C 180,E1 -22003.737,E2 -22003.737} C_VEL
LIN {X 0,Y 223.938,Z 425.84,A -85,B 0,C 180,E1 -22005.59,E2 -22005.59} C_VEL
LIN {X 0,Y 222.345,Z 439.727,A -85,B 0,C 180,E1 -22007.694,E2 -22007.694} C_VEL
LIN {X 0,Y 220.406,Z 451.63,A -85,B 0,C 180,E1 -22009.782,E2 -22009.782} C_VEL
LIN {X 0,Y 215.973,Z 463.406,A -85,B 0,C 180,E1 -22011.81,E2 -22011.81} C_VEL
LIN {X 0,Y 211.024,Z 475.244,A -85,B 0,C 180,E1 -22014.351,E2 -22014.351} C_VEL
LIN {X 0,Y 206.57,Z 485.225,A -85,B 0,C 180,E1 -22017.02,E2 -22017.02} C_VEL
LIN {X 0,Y 204.163,Z 490.53,A -85,B 0,C 180,E1 -22018.702,E2 -22018.702} C_VEL
LIN {X 0,Y 202.419,Z 492.972,A -85,B 0,C 180,E1 -22019.458,E2 -22019.458} C_VEL
LIN {X 0,Y 193.769,Z 500.046,A -85,B 0,C 180,E1 -22021.646,E2 -22021.646} C_VEL
LIN {X 0,Y 192.179,Z 502.117,A -85,B 0,C 180,E1 -22022.537,E2 -22022.537} C_VEL
LIN {X 0,Y 189.148,Z 508.48,A -85,B 0,C 180,E1 -22025.876,E2 -22025.876} C_VEL
LIN {X 0,Y 186.341,Z 514.967,A -85,B 0,C 180,E1 -22030.158,E2 -22030.158} C_VEL
LIN {X 0,Y 184.527,Z 520.016,A -85,B 0,C 180,E1 -22034.538,E2 -22034.538} C_VEL
LIN {X 0,Y 183.693,Z 523.754,A -85,B 0,C 180,E1 -22038.972,E2 -22038.972} C_VEL
LIN {X 0,Y 183.796,Z 526.429,A -85,B 0,C 180,E1 -22043.818,E2 -22043.818} C_VEL
LIN {X 0,Y 184.024,Z 527.547,A -85,B 0,C 180,E1 -22047.812,E2 -22047.812} C_VEL
LIN {X 0,Y 184.363,Z 527.738,A -85,B 0,C 180,E1 -22050,E2 -22050} C_VEL
LIN {X 0,Y 183.905,Z 527.053,A -85,B 0,C 180,E1 -22054.384,E2 -22054.384} C_VEL
LIN {X 0,Y 183.736,Z 526.249,A -85,B 0,C 180,E1 -22056.59,E2 -22056.59} C_VEL
LIN {X 0,Y 183.707,Z 523.723,A -85,B 0,C 180,E1 -22061.028,E2 -22061.028} C_VEL
LIN {X 0,Y 184.549,Z 519.961,A -85,B 0,C 180,E1 -22065.461,E2 -22065.461} C_VEL
LIN {X 0,Y 186.346,Z 514.889,A -85,B 0,C 180,E1 -22069.843,E2 -22069.843} C_VEL
LIN {X 0,Y 189.154,Z 508.389,A -85,B 0,C 180,E1 -22074.124,E2 -22074.124} C_VEL
LIN {X 0,Y 193.078,Z 500.28,A -85,B 0,C 180,E1 -22078.243,E2 -22078.243} C_VEL
LIN {X 0,Y 196.172,Z 494.102,A -85,B 0,C 180,E1 -22080.908,E2 -22080.908} C_VEL
LIN {X 0,Y 202.58,Z 489.226,A -85,B 0,C 180,E1 -22084.92,E2 -22084.92} C_VEL
LIN {X 0,Y 211.582,Z 482.436,A -85,B 0,C 180,E1 -22089.133,E2 -22089.133} C_VEL
LIN {X 0,Y 220.004,Z 476.062,A -85,B 0,C 180,E1 -22092.133,E2 -22092.133} C_VEL
LIN {X 0,Y 231.821,Z 466.842,A -85,B 0,C 180,E1 -22095.434,E2 -22095.434} C_VEL
LIN {X 0,Y 239.013,Z 460.72,A -85,B 0,C 180,E1 -22097.317,E2 -22097.317} C_VEL
LIN {X 0,Y 243.578,Z 456.659,A -85,B 0,C 180,E1 -22098.607,E2 -22098.607} C_VEL
LIN {X 0,Y 245.551,Z 454.685,A -85,B 0,C 180,E1 -22099.33,E2 -22099.33} C_VEL
LIN {X 0,Y 246.107,Z 453.58,A -85,B 0,C 180,E1 -22100.447,E2 -22100.447} C_VEL
LIN {X 0,Y 245.719,Z 453.043,A -85,B 0,C 180,E1 -22102.053,E2 -22102.053} C_VEL
LIN {X 0,Y 244.111,Z 453.829,A -85,B 0,C 180,E1 -22102.801,E2 -22102.801} C_VEL
LIN {X 0,Y 234.642,Z 458.976,A -85,B 0,C 180,E1 -22105.314,E2 -22105.314} C_VEL
LIN {X 0,Y 225.878,Z 462.952,A -85,B 0,C 180,E1 -22108.066,E2 -22108.066} C_VEL
LIN {X 0,Y 217.798,Z 465.829,A -85,B 0,C 180,E1 -22111.052,E2 -22111.052} C_VEL
LIN {X 0,Y 210.497,Z 467.596,A -85,B 0,C 180,E1 -22114.276,E2 -22114.276} C_VEL
LIN {X 0,Y 204.099,Z 468.234,A -85,B 0,C 180,E1 -22117.742,E2 -22117.742} C_VEL
LIN {X 0,Y 198.564,Z 467.755,A -85,B 0,C 180,E1 -22121.425,E2 -22121.425} C_VEL
LIN {X 0,Y 194.008,Z 466.077,A -85,B 0,C 180,E1 -22125.311,E2 -22125.311} C_VEL
LIN {X 0,Y 190.514,Z 463.141,A -85,B 0,C 180,E1 -22129.371,E2 -22129.371} C_VEL
LIN {X 0,Y 188.089,Z 458.92,A -85,B 0,C 180,E1 -22133.564,E2 -22133.564} C_VEL
LIN {X 0,Y 186.372,Z 453.254,A -85,B 0,C 180,E1 -22137.839,E2 -22137.839} C_VEL
LIN {X 0,Y 185.46,Z 446.058,A -85,B 0,C 180,E1 -22142.172,E2 -22142.172} C_VEL
LIN {X 0,Y 185.399,Z 438.315,A -85,B 0,C 180,E1 -22145.984,E2 -22145.984} C_VEL
LIN {X 0,Y 186.182,Z 428.994,A -85,B 0,C 180,E1 -22149.78,E2 -22149.78} C_VEL
LIN {X 0,Y 187.299,Z 417.656,A -85,B 0,C 180,E1 -22153.563,E2 -22153.563} C_VEL
LIN {X 0,Y 188.513,Z 405.98,A -85,B 0,C 180,E1 -22156.794,E2 -22156.794} C_VEL
LIN {X 0,Y 190.297,Z 392.015,A -85,B 0,C 180,E1 -22159.976,E2 -22159.976} C_VEL
LIN {X 0,Y 191.939,Z 379.463,A -85,B 0,C 180,E1 -22162.327,E2 -22162.327} C_VEL
LIN {X 0,Y 192.95,Z 369.179,A -85,B 0,C 180,E1 -22163.95,E2 -22163.95} C_VEL
LIN {X 0,Y 190.33,Z 356.842,A -85,B 0,C 180,E1 -22165.837,E2 -22165.837} C_VEL
LIN {X 0,Y 190.827,Z 357.541,A -85,B 0,C 180,E1 -22166.229,E2 -22166.229} C_VEL
LIN {X 0,Y 192.078,Z 357.205,A -85,B 0,C 180,E1 -22166.964,E2 -22166.964} C_VEL
LIN {X 0,Y 193.686,Z 355.161,A -85,B 0,C 180,E1 -22167.705,E2 -22167.705} C_VEL
LIN {X 0,Y 194.492,Z 353.674,A -85,B 0,C 180,E1 -22168.019,E2 -22168.019} C_VEL
LIN {X 0,Y 195.088,Z 353.77,A -85,B 0,C 180,E1 -22168.365,E2 -22168.365} C_VEL
LIN {X 0,Y 199.222,Z 357.825,A -85,B 0,C 180,E1 -22170.912,E2 -22170.912} C_VEL
LIN {X 0,Y 202.478,Z 361.76,A -85,B 0,C 180,E1 -22172.844,E2 -22172.844} C_VEL
LIN {X 0,Y 206.253,Z 367.41,A -85,B 0,C 180,E1 -22175.084,E2 -22175.084} C_VEL
LIN {X 0,Y 210.274,Z 374.03,A -85,B 0,C 180,E1 -22177.468,E2 -22177.468} C_VEL
LIN {X 0,Y 214.648,Z 383.173,A -85,B 0,C 180,E1 -22180.29,E2 -22180.29} C_VEL
LIN {X 0,Y 217.107,Z 389.957,A -85,B 0,C 180,E1 -22182.137,E2 -22182.137} C_VEL
LIN {X 0,Y 219.792,Z 400.201,A -85,B 0,C 180,E1 -22184.706,E2 -22184.706} C_VEL
LIN {X 0,Y 221.451,Z 410.197,A -85,B 0,C 180,E1 -22187.157,E2 -22187.157} C_VEL
LIN {X 0,Y 221.884,Z 414.98,A -85,B 0,C 180,E1 -22188.305,E2 -22188.305} C_VEL
LIN {X 0,Y 217.445,Z 427.76,A -85,B 0,C 180,E1 -22190.332,E2 -22190.332} C_VEL
LIN {X 0,Y 212.979,Z 438.999,A -85,B 0,C 180,E1 -22192.539,E2 -22192.539} C_VEL
LIN {X 0,Y 208.603,Z 449.278,A -85,B 0,C 180,E1 -22195.058,E2 -22195.058} C_VEL
LIN {X 0,Y 204.23,Z 458.372,A -85,B 0,C 180,E1 -22197.765,E2 -22197.765} C_VEL
LIN {X 0,Y 199.672,Z 467.279,A -85,B 0,C 180,E1 -22201.054,E2 -22201.054} C_VEL
LIN {X 0,Y 195.698,Z 474.655,A -85,B 0,C 180,E1 -22204.472,E2 -22204.472} C_VEL
LIN {X 0,Y 191.883,Z 481.515,A -85,B 0,C 180,E1 -22208.514,E2 -22208.514} C_VEL
LIN {X 0,Y 188.939,Z 486.884,A -85,B 0,C 180,E1 -22212.687,E2 -22212.687} C_VEL
LIN {X 0,Y 186.73,Z 490.934,A -85,B 0,C 180,E1 -22216.948,E2 -22216.948} C_VEL
LIN {X 0,Y 185.265,Z 493.766,A -85,B 0,C 180,E1 -22221.272,E2 -22221.272} C_VEL
LIN {X 0,Y 184.62,Z 495.44,A -85,B 0,C 180,E1 -22225.633,E2 -22225.633} C_VEL
LIN {X 0,Y 184.351,Z 496.024,A -85,B 0,C 180,E1 -22230,E2 -22230} C_VEL
LIN {X 0,Y 184.584,Z 495.472,A -85,B 0,C 180,E1 -22234.367,E2 -22234.367} C_VEL
LIN {X 0,Y 185.266,Z 493.834,A -85,B 0,C 180,E1 -22238.727,E2 -22238.727} C_VEL
LIN {X 0,Y 186.725,Z 491.05,A -85,B 0,C 180,E1 -22243.051,E2 -22243.051} C_VEL
LIN {X 0,Y 188.893,Z 487.054,A -85,B 0,C 180,E1 -22247.316,E2 -22247.316} C_VEL
LIN {X 0,Y 191.827,Z 481.73,A -85,B 0,C 180,E1 -22251.492,E2 -22251.492} C_VEL
LIN {X 0,Y 195.631,Z 474.916,A -85,B 0,C 180,E1 -22255.537,E2 -22255.537} C_VEL
LIN {X 0,Y 199.575,Z 467.603,A -85,B 0,C 180,E1 -22258.96,E2 -22258.96} C_VEL
LIN {X 0,Y 204.135,Z 458.765,A -85,B 0,C 180,E1 -22262.251,E2 -22262.251} C_VEL
LIN {X 0,Y 208.496,Z 449.706,A -85,B 0,C 180,E1 -22264.962,E2 -22264.962} C_VEL
LIN {X 0,Y 213.335,Z 438.347,A -85,B 0,C 180,E1 -22267.754,E2 -22267.754} C_VEL
LIN {X 0,Y 218.225,Z 426.092,A -85,B 0,C 180,E1 -22270.098,E2 -22270.098} C_VEL
LIN {X 0,Y 222.033,Z 414.354,A -85,B 0,C 180,E1 -22271.964,E2 -22271.964} C_VEL
LIN {X 0,Y 220.552,Z 404.004,A -85,B 0,C 180,E1 -22274.51,E2 -22274.51} C_VEL
LIN {X 0,Y 218.523,Z 394.507,A -85,B 0,C 180,E1 -22276.853,E2 -22276.853} C_VEL
LIN {X 0,Y 215.547,Z 385.211,A -85,B 0,C 180,E1 -22279.299,E2 -22279.299} C_VEL
LIN {X 0,Y 211.159,Z 375.818,A -85,B 0,C 180,E1 -22282.158,E2 -22282.158} C_VEL
LIN {X 0,Y 207.362,Z 369.111,A -85,B 0,C 180,E1 -22284.463,E2 -22284.463} C_VEL
LIN {X 0,Y 204.662,Z 364.866,A -85,B 0,C 180,E1 -22286.081,E2 -22286.081} C_VEL
LIN {X 0,Y 202.14,Z 361.039,A -85,B 0,C 180,E1 -22287.612,E2 -22287.612} C_VEL
LIN {X 0,Y 199.474,Z 357.268,A -85,B 0,C 180,E1 -22289.245,E2 -22289.245} C_VEL
LIN {X 0,Y 195.946,Z 353.015,A -85,B 0,C 180,E1 -22291.479,E2 -22291.479} C_VEL
LIN {X 0,Y 194.913,Z 351.508,A -85,B 0,C 180,E1 -22292.177,E2 -22292.177} C_VEL
LIN {X 0,Y 191.918,Z 348.445,A -85,B 0,C 180,E1 -22294.223,E2 -22294.223} C_VEL
LIN {X 0,Y 190.769,Z 346.373,A -85,B 0,C 180,E1 -22295.225,E2 -22295.225} C_VEL
LIN {X 0,Y 190.61,Z 344.913,A -85,B 0,C 180,E1 -22298.364,E2 -22298.364} C_VEL
LIN {X 0,Y 190.32,Z 343.008,A -85,B 0,C 180,E1 -22303.761,E2 -22303.761} C_VEL
LIN {X 0,Y 190.302,Z 341.673,A -85,B 0,C 180,E1 -22309.359,E2 -22309.359} C_VEL
LIN {X 0,Y 190.407,Z 341.285,A -85,B 0,C 180,E1 -22311.509,E2 -22311.509} C_VEL
LIN {X 0,Y 190.627,Z 340.922,A -85,B 0,C 180,E1 -22317.887,E2 -22317.887} C_VEL
LIN {X 0,Y 190.879,Z 340.981,A -85,B 0,C 180,E1 -22320,E2 -22320} C_VEL
LIN {X 0,Y 190.918,Z 341.91,A -85,B 0,C 180,E1 -22324.222,E2 -22324.222} C_VEL
LIN {X 0,Y 191.556,Z 343.151,A -85,B 0,C 180,E1 -22328.439,E2 -22328.439} C_VEL
LIN {X 0,Y 192.146,Z 345.18,A -85,B 0,C 180,E1 -22332.677,E2 -22332.677} C_VEL
LIN {X 0,Y 193.24,Z 347.69,A -85,B 0,C 180,E1 -22336.915,E2 -22336.915} C_VEL
LIN {X 0,Y 194.472,Z 351.044,A -85,B 0,C 180,E1 -22341.185,E2 -22341.185} C_VEL
LIN {X 0,Y 196.83,Z 356.456,A -85,B 0,C 180,E1 -22346.793,E2 -22346.793} C_VEL
LIN {X 0,Y 197.46,Z 359.233,A -85,B 0,C 180,E1 -22348.863,E2 -22348.863} C_VEL
LIN {X 0,Y 200.1,Z 364.093,A -85,B 0,C 180,E1 -22350.514,E2 -22350.514} C_VEL
LIN {X 0,Y 201.536,Z 366.427,A -85,B 0,C 180,E1 -22351.343,E2 -22351.343} C_VEL
LIN {X 0,Y 204.593,Z 371.724,A -85,B 0,C 180,E1 -22353.047,E2 -22353.047} C_VEL
LIN {X 0,Y 208.512,Z 379.265,A -85,B 0,C 180,E1 -22355.18,E2 -22355.18} C_VEL
LIN {X 0,Y 213.232,Z 389.26,A -85,B 0,C 180,E1 -22357.785,E2 -22357.785} C_VEL
LIN {X 0,Y 217.199,Z 399.051,A -85,B 0,C 180,E1 -22360.099,E2 -22360.099} C_VEL
LIN {X 0,Y 218.983,Z 403.556,A -85,B 0,C 180,E1 -22361.141,E2 -22361.141} C_VEL
LIN {X 0,Y 219.135,Z 416.958,A -85,B 0,C 180,E1 -22363.025,E2 -22363.025} C_VEL
LIN {X 0,Y 218.031,Z 430.726,A -85,B 0,C 180,E1 -22365.035,E2 -22365.035} C_VEL
LIN {X 0,Y 216.029,Z 444.119,A -85,B 0,C 180,E1 -22367.226,E2 -22367.226} C_VEL
LIN {X 0,Y 214.091,Z 453.621,A -85,B 0,C 180,E1 -22368.964,E2 -22368.964} C_VEL
LIN {X 0,Y 208.699,Z 467.032,A -85,B 0,C 180,E1 -22371.466,E2 -22371.466} C_VEL
LIN {X 0,Y 203.595,Z 478.181,A -85,B 0,C 180,E1 -22374.068,E2 -22374.068} C_VEL
LIN {X 0,Y 199.143,Z 487.621,A -85,B 0,C 180,E1 -22376.838,E2 -22376.838} C_VEL
LIN {X 0,Y 194.753,Z 496.677,A -85,B 0,C 180,E1 -22380.143,E2 -22380.143} C_VEL
LIN {X 0,Y 192.179,Z 502.117,A -85,B 0,C 180,E1 -22382.537,E2 -22382.537} C_VEL
LIN {X 0,Y 190.189,Z 505.089,A -85,B 0,C 180,E1 -22383.955,E2 -22383.955} C_VEL
LIN {X 0,Y 185.311,Z 509.517,A -85,B 0,C 180,E1 -22386.227,E2 -22386.227} C_VEL
LIN {X 0,Y 180.659,Z 513.406,A -85,B 0,C 180,E1 -22388.684,E2 -22388.684} C_VEL
LIN {X 0,Y 179.069,Z 515.575,A -85,B 0,C 180,E1 -22390.352,E2 -22390.352} C_VEL
LIN {X 0,Y 177.274,Z 520.483,A -85,B 0,C 180,E1 -22395.067,E2 -22395.067} C_VEL
LIN {X 0,Y 176.632,Z 523.136,A -85,B 0,C 180,E1 -22398.525,E2 -22398.525} C_VEL
LIN {X 0,Y 176.625,Z 525.65,A -85,B 0,C 180,E1 -22403.145,E2 -22403.145} C_VEL
LIN {X 0,Y 176.816,Z 526.451,A -85,B 0,C 180,E1 -22405.441,E2 -22405.441} C_VEL
LIN {X 0,Y 177.285,Z 527.13,A -85,B 0,C 180,E1 -22410.001,E2 -22410.001} C_VEL
LIN {X 0,Y 176.831,Z 526.442,A -85,B 0,C 180,E1 -22414.56,E2 -22414.56} C_VEL
LIN {X 0,Y 176.536,Z 524.52,A -85,B 0,C 180,E1 -22419.163,E2 -22419.163} C_VEL
LIN {X 0,Y 176.993,Z 521.379,A -85,B 0,C 180,E1 -22423.784,E2 -22423.784} C_VEL
LIN {X 0,Y 178.481,Z 516.976,A -85,B 0,C 180,E1 -22428.362,E2 -22428.362} C_VEL
LIN {X 0,Y 180.929,Z 511.205,A -85,B 0,C 180,E1 -22432.858,E2 -22432.858} C_VEL
LIN {X 0,Y 184.579,Z 503.935,A -85,B 0,C 180,E1 -22437.189,E2 -22437.189} C_VEL
LIN {X 0,Y 188.85,Z 495.442,A -85,B 0,C 180,E1 -22441.137,E2 -22441.137} C_VEL
LIN {X 0,Y 189.813,Z 493.805,A -85,B 0,C 180,E1 -22441.845,E2 -22441.845} C_VEL
LIN {X 0,Y 198.529,Z 487.957,A -85,B 0,C 180,E1 -22447,E2 -22447} C_VEL
LIN {X 0,Y 206.144,Z 482.776,A -85,B 0,C 180,E1 -22450.374,E2 -22450.374} C_VEL
LIN {X 0,Y 214.837,Z 476.852,A -85,B 0,C 180,E1 -22453.392,E2 -22453.392} C_VEL
LIN {X 0,Y 226.976,Z 468.215,A -85,B 0,C 180,E1 -22456.69,E2 -22456.69} C_VEL
LIN {X 0,Y 234.421,Z 462.517,A -85,B 0,C 180,E1 -22458.548,E2 -22458.548} C_VEL
LIN {X 0,Y 239.125,Z 458.685,A -85,B 0,C 180,E1 -22459.832,E2 -22459.832} C_VEL
LIN {X 0,Y 240.14,Z 457.274,A -85,B 0,C 180,E1 -22461.065,E2 -22461.065} C_VEL
LIN {X 0,Y 239.057,Z 457.546,A -85,B 0,C 180,E1 -22461.875,E2 -22461.875} C_VEL
LIN {X 0,Y 229.334,Z 462.179,A -85,B 0,C 180,E1 -22464.391,E2 -22464.391} C_VEL
LIN {X 0,Y 220.27,Z 465.709,A -85,B 0,C 180,E1 -22467.153,E2 -22467.153} C_VEL
LIN {X 0,Y 211.929,Z 468.17,A -85,B 0,C 180,E1 -22470.17,E2 -22470.17} C_VEL
LIN {X 0,Y 203.596,Z 469.614,A -85,B 0,C 180,E1 -22473.833,E2 -22473.833} C_VEL
LIN {X 0,Y 197.719,Z 469.829,A -85,B 0,C 180,E1 -22476.984,E2 -22476.984} C_VEL
LIN {X 0,Y 191.949,Z 468.989,A -85,B 0,C 180,E1 -22480.76,E2 -22480.76} C_VEL
LIN {X 0,Y 187.215,Z 466.952,A -85,B 0,C 180,E1 -22484.765,E2 -22484.765} C_VEL
LIN {X 0,Y 183.584,Z 463.671,A -85,B 0,C 180,E1 -22488.965,E2 -22488.965} C_VEL
LIN {X 0,Y 181.055,Z 459.098,A -85,B 0,C 180,E1 -22493.313,E2 -22493.313} C_VEL
LIN {X 0,Y 179.263,Z 453.143,A -85,B 0,C 180,E1 -22497.753,E2 -22497.753} C_VEL
LIN {X 0,Y 178.354,Z 445.615,A -85,B 0,C 180,E1 -22502.259,E2 -22502.259} C_VEL
LIN {X 0,Y 178.334,Z 437.53,A -85,B 0,C 180,E1 -22506.222,E2 -22506.222} C_VEL
LIN {X 0,Y 179.079,Z 429.362,A -85,B 0,C 180,E1 -22509.602,E2 -22509.602} C_VEL
LIN {X 0,Y 180.16,Z 417.985,A -85,B 0,C 180,E1 -22513.536,E2 -22513.536} C_VEL
LIN {X 0,Y 181.416,Z 406.175,A -85,B 0,C 180,E1 -22516.891,E2 -22516.891} C_VEL
LIN {X 0,Y 183.22,Z 392.043,A -85,B 0,C 180,E1 -22520.196,E2 -22520.196} C_VEL
LIN {X 0,Y 184.913,Z 379.29,A -85,B 0,C 180,E1 -22522.633,E2 -22522.633} C_VEL
LIN {X 0,Y 185.897,Z 371.113,A -85,B 0,C 180,E1 -22523.98,E2 -22523.98} C_VEL
LIN {X 0,Y 185.717,Z 369.072,A -85,B 0,C 180,E1 -22524.376,E2 -22524.376} C_VEL
LIN {X 0,Y 185.905,Z 369.48,A -85,B 0,C 180,E1 -22524.573,E2 -22524.573} C_VEL
LIN {X 0,Y 187.459,Z 369.431,A -85,B 0,C 180,E1 -22525.631,E2 -22525.631} C_VEL
LIN {X 0,Y 189.37,Z 367.136,A -85,B 0,C 180,E1 -22526.532,E2 -22526.532} C_VEL
LIN {X 0,Y 190.913,Z 364.424,A -85,B 0,C 180,E1 -22527.112,E2 -22527.112} C_VEL
LIN {X 0,Y 192.8,Z 363.26,A -85,B 0,C 180,E1 -22528.077,E2 -22528.077} C_VEL
LIN {X 0,Y 193.644,Z 362.389,A -85,B 0,C 180,E1 -22528.448,E2 -22528.448} C_VEL
LIN {X 0,Y 195.056,Z 362.558,A -85,B 0,C 180,E1 -22529.253,E2 -22529.253} C_VEL
LIN {X 0,Y 196.718,Z 364.246,A -85,B 0,C 180,E1 -22530.341,E2 -22530.341} C_VEL
LIN {X 0,Y 200.183,Z 368.862,A -85,B 0,C 180,E1 -22532.608,E2 -22532.608} C_VEL
LIN {X 0,Y 202.744,Z 372.905,A -85,B 0,C 180,E1 -22534.296,E2 -22534.296} C_VEL
LIN {X 0,Y 206.564,Z 379.701,A -85,B 0,C 180,E1 -22536.846,E2 -22536.846} C_VEL
LIN {X 0,Y 210.73,Z 389.19,A -85,B 0,C 180,E1 -22539.908,E2 -22539.908} C_VEL
LIN {X 0,Y 212.837,Z 396.153,A -85,B 0,C 180,E1 -22541.855,E2 -22541.855} C_VEL
LIN {X 0,Y 215.085,Z 406.695,A -85,B 0,C 180,E1 -22544.629,E2 -22544.629} C_VEL
LIN {X 0,Y 216.194,Z 416.964,A -85,B 0,C 180,E1 -22547.265,E2 -22547.265} C_VEL
LIN {X 0,Y 211.577,Z 429.507,A -85,B 0,C 180,E1 -22549.315,E2 -22549.315} C_VEL
LIN {X 0,Y 207.303,Z 439.847,A -85,B 0,C 180,E1 -22551.407,E2 -22551.407} C_VEL
LIN {X 0,Y 202.846,Z 449.883,A -85,B 0,C 180,E1 -22553.913,E2 -22553.913} C_VEL
LIN {X 0,Y 198.287,Z 458.977,A -85,B 0,C 180,E1 -22556.675,E2 -22556.675} C_VEL
LIN {X 0,Y 193.511,Z 467.886,A -85,B 0,C 180,E1 -22560.041,E2 -22560.041} C_VEL
LIN {X 0,Y 189.327,Z 475.264,A -85,B 0,C 180,E1 -22563.547,E2 -22563.547} C_VEL
LIN {X 0,Y 185.294,Z 482.125,A -85,B 0,C 180,E1 -22567.71,E2 -22567.71} C_VEL
LIN {X 0,Y 182.187,Z 487.494,A -85,B 0,C 180,E1 -22572.024,E2 -22572.024} C_VEL
LIN {X 0,Y 179.845,Z 491.543,A -85,B 0,C 180,E1 -22576.439,E2 -22576.439} C_VEL
LIN {X 0,Y 178.287,Z 494.374,A -85,B 0,C 180,E1 -22580.927,E2 -22580.927} C_VEL
LIN {X 0,Y 177.554,Z 496.05,A -85,B 0,C 180,E1 -22585.459,E2 -22585.459} C_VEL
LIN {X 0,Y 177.29,Z 496.631,A -85,B 0,C 180,E1 -22589.999,E2 -22589.999} C_VEL
LIN {X 0,Y 177.519,Z 496.081,A -85,B 0,C 180,E1 -22594.541,E2 -22594.541} C_VEL
LIN {X 0,Y 178.287,Z 494.441,A -85,B 0,C 180,E1 -22599.072,E2 -22599.072} C_VEL
LIN {X 0,Y 179.84,Z 491.657,A -85,B 0,C 180,E1 -22603.56,E2 -22603.56} C_VEL
LIN {X 0,Y 182.143,Z 487.662,A -85,B 0,C 180,E1 -22607.979,E2 -22607.979} C_VEL
LIN {X 0,Y 185.24,Z 482.338,A -85,B 0,C 180,E1 -22612.296,E2 -22612.296} C_VEL
LIN {X 0,Y 189.27,Z 475.521,A -85,B 0,C 180,E1 -22616.46,E2 -22616.46} C_VEL
LIN {X 0,Y 193.394,Z 468.209,A -85,B 0,C 180,E1 -22619.978,E2 -22619.978} C_VEL
LIN {X 0,Y 198.179,Z 459.367,A -85,B 0,C 180,E1 -22623.344,E2 -22623.344} C_VEL
LIN {X 0,Y 202.723,Z 450.308,A -85,B 0,C 180,E1 -22626.111,E2 -22626.111} C_VEL
LIN {X 0,Y 207.64,Z 439.26,A -85,B 0,C 180,E1 -22628.878,E2 -22628.878} C_VEL
LIN {X 0,Y 212.865,Z 426.685,A -85,B 0,C 180,E1 -22631.324,E2 -22631.324} C_VEL
LIN {X 0,Y 216.053,Z 417.701,A -85,B 0,C 180,E1 -22632.768,E2 -22632.768} C_VEL
LIN {X 0,Y 216.301,Z 416.337,A -85,B 0,C 180,E1 -22633.025,E2 -22633.025} C_VEL
LIN {X 0,Y 214.778,Z 404.681,A -85,B 0,C 180,E1 -22636.045,E2 -22636.045} C_VEL
LIN {X 0,Y 212.612,Z 395.042,A -85,B 0,C 180,E1 -22638.615,E2 -22638.615} C_VEL
LIN {X 0,Y 210.347,Z 388.202,A -85,B 0,C 180,E1 -22640.593,E2 -22640.593} C_VEL
LIN {X 0,Y 206.036,Z 378.673,A -85,B 0,C 180,E1 -22643.715,E2 -22643.715} C_VEL
LIN {X 0,Y 203.438,Z 374.037,A -85,B 0,C 180,E1 -22645.474,E2 -22645.474} C_VEL
LIN {X 0,Y 199.377,Z 367.196,A -85,B 0,C 180,E1 -22648.228,E2 -22648.228} C_VEL
LIN {X 0,Y 196.044,Z 362.509,A -85,B 0,C 180,E1 -22650.467,E2 -22650.467} C_VEL
LIN {X 0,Y 193.27,Z 358.736,A -85,B 0,C 180,E1 -22652.435,E2 -22652.435} C_VEL
LIN {X 0,Y 192.225,Z 357.49,A -85,B 0,C 180,E1 -22653.184,E2 -22653.184} C_VEL
LIN {X 0,Y 189.516,Z 354.214,A -85,B 0,C 180,E1 -22655.269,E2 -22655.269} C_VEL
LIN {X 0,Y 188.548,Z 352.817,A -85,B 0,C 180,E1 -22656.066,E2 -22656.066} C_VEL
LIN {X 0,Y 185.275,Z 349.494,A -85,B 0,C 180,E1 -22658.877,E2 -22658.877} C_VEL
LIN {X 0,Y 184.208,Z 347.628,A -85,B 0,C 180,E1 -22660.063,E2 -22660.063} C_VEL
LIN {X 0,Y 184.079,Z 346.219,A -85,B 0,C 180,E1 -22664.499,E2 -22664.499} C_VEL
LIN {X 0,Y 184.153,Z 345.311,A -85,B 0,C 180,E1 -22668.999,E2 -22668.999} C_VEL
LIN {X 0,Y 184.218,Z 344.776,A -85,B 0,C 180,E1 -22672.705,E2 -22672.705} C_VEL
LIN {X 0,Y 184.568,Z 344.664,A -85,B 0,C 180,E1 -22677.818,E2 -22677.818} C_VEL
LIN {X 0,Y 184.879,Z 344.755,A -85,B 0,C 180,E1 -22680,E2 -22680} C_VEL
LIN {X 0,Y 184.99,Z 345.811,A -85,B 0,C 180,E1 -22684.357,E2 -22684.357} C_VEL
LIN {X 0,Y 185.663,Z 347.185,A -85,B 0,C 180,E1 -22688.709,E2 -22688.709} C_VEL
LIN {X 0,Y 186.323,Z 349.352,A -85,B 0,C 180,E1 -22693.08,E2 -22693.08} C_VEL
LIN {X 0,Y 187.465,Z 352.063,A -85,B 0,C 180,E1 -22697.452,E2 -22697.452} C_VEL
LIN {X 0,Y 189.207,Z 356.554,A -85,B 0,C 180,E1 -22702.955,E2 -22702.955} C_VEL
LIN {X 0,Y 189.883,Z 358.064,A -85,B 0,C 180,E1 -22704.388,E2 -22704.388} C_VEL
LIN {X 0,Y 194.994,Z 365.377,A -85,B 0,C 180,E1 -22708.013,E2 -22708.013} C_VEL
LIN {X 0,Y 197.953,Z 370.697,A -85,B 0,C 180,E1 -22709.951,E2 -22709.951} C_VEL
LIN {X 0,Y 202.468,Z 379.416,A -85,B 0,C 180,E1 -22712.771,E2 -22712.771} C_VEL
LIN {X 0,Y 204.794,Z 384.149,A -85,B 0,C 180,E1 -22714.198,E2 -22714.198} C_VEL
LIN {X 0,Y 209.015,Z 393.736,A -85,B 0,C 180,E1 -22716.82,E2 -22716.82} C_VEL
LIN {X 0,Y 212.295,Z 402.299,A -85,B 0,C 180,E1 -22718.976,E2 -22718.976} C_VEL
LIN {X 0,Y 213.985,Z 407.143,A -85,B 0,C 180,E1 -22720.163,E2 -22720.163} C_VEL
LIN {X 0,Y 213.687,Z 420.886,A -85,B 0,C 180,E1 -22722.19,E2 -22722.19} C_VEL
LIN {X 0,Y 212.093,Z 434.855,A -85,B 0,C 180,E1 -22724.36,E2 -22724.36} C_VEL
LIN {X 0,Y 209.775,Z 447.743,A -85,B 0,C 180,E1 -22726.623,E2 -22726.623} C_VEL
LIN {X 0,Y 208.321,Z 454.081,A -85,B 0,C 180,E1 -22727.855,E2 -22727.855} C_VEL
LIN {X 0,Y 203.115,Z 466.424,A -85,B 0,C 180,E1 -22730.2,E2 -22730.2} C_VEL
LIN {X 0,Y 197.828,Z 477.572,A -85,B 0,C 180,E1 -22732.848,E2 -22732.848} C_VEL
LIN {X 0,Y 193.172,Z 487.01,A -85,B 0,C 180,E1 -22735.673,E2 -22735.673} C_VEL
LIN {X 0,Y 188.182,Z 496.766,A -85,B 0,C 180,E1 -22739.339,E2 -22739.339} C_VEL
LIN {X 0,Y 184.534,Z 504.035,A -85,B 0,C 180,E1 -22742.805,E2 -22742.805} C_VEL
LIN {X 0,Y 180.931,Z 511.293,A -85,B 0,C 180,E1 -22747.143,E2 -22747.143} C_VEL
LIN {X 0,Y 179.069,Z 515.575,A -85,B 0,C 180,E1 -22750.352,E2 -22750.352} C_VEL
LIN {X 0,Y 177.627,Z 517.595,A -85,B 0,C 180,E1 -22752.073,E2 -22752.073} C_VEL
LIN {X 0,Y 173.76,Z 520.3,A -85,B 0,C 180,E1 -22754.918,E2 -22754.918} C_VEL
LIN {X 0,Y 170.811,Z 522.091,A -85,B 0,C 180,E1 -22757.31,E2 -22757.31} C_VEL
LIN {X 0,Y 169.562,Z 523.279,A -85,B 0,C 180,E1 -22759.221,E2 -22759.221} C_VEL
LIN {X 0,Y 169.45,Z 523.59,A -85,B 0,C 180,E1 -22759.875,E2 -22759.875} C_VEL
LIN {X 0,Y 169.638,Z 525.415,A -85,B 0,C 180,E1 -22763.882,E2 -22763.882} C_VEL
LIN {X 0,Y 169.848,Z 526.327,A -85,B 0,C 180,E1 -22767.629,E2 -22767.629} C_VEL
LIN {X 0,Y 170.209,Z 526.521,A -85,B 0,C 180,E1 -22770.001,E2 -22770.001} C_VEL
LIN {X 0,Y 169.732,Z 525.83,A -85,B 0,C 180,E1 -22774.751,E2 -22774.751} C_VEL
LIN {X 0,Y 169.455,Z 523.902,A -85,B 0,C 180,E1 -22779.55,E2 -22779.55} C_VEL
LIN {X 0,Y 170.017,Z 520.76,A -85,B 0,C 180,E1 -22784.361,E2 -22784.361} C_VEL
LIN {X 0,Y 171.635,Z 516.354,A -85,B 0,C 180,E1 -22789.123,E2 -22789.123} C_VEL
LIN {X 0,Y 174.301,Z 510.584,A -85,B 0,C 180,E1 -22793.78,E2 -22793.78} C_VEL
LIN {X 0,Y 178.206,Z 503.316,A -85,B 0,C 180,E1 -22798.246,E2 -22798.246} C_VEL
LIN {X 0,Y 182.35,Z 495.52,A -85,B 0,C 180,E1 -22802.016,E2 -22802.016} C_VEL
LIN {X 0,Y 183.759,Z 493.202,A -85,B 0,C 180,E1 -22803.025,E2 -22803.025} C_VEL
LIN {X 0,Y 192.863,Z 487.81,A -85,B 0,C 180,E1 -22808.279,E2 -22808.279} C_VEL
LIN {X 0,Y 200.787,Z 483.046,A -85,B 0,C 180,E1 -22811.686,E2 -22811.686} C_VEL
LIN {X 0,Y 212.192,Z 476.015,A -85,B 0,C 180,E1 -22815.407,E2 -22815.407} C_VEL
LIN {X 0,Y 224.856,Z 467.741,A -85,B 0,C 180,E1 -22818.603,E2 -22818.603} C_VEL
LIN {X 0,Y 231.329,Z 463.143,A -85,B 0,C 180,E1 -22820.201,E2 -22820.201} C_VEL
LIN {X 0,Y 233.595,Z 461.472,A -85,B 0,C 180,E1 -22820.816,E2 -22820.816} C_VEL
LIN {X 0,Y 228.946,Z 463.359,A -85,B 0,C 180,E1 -22822.125,E2 -22822.125} C_VEL
LIN {X 0,Y 219.315,Z 466.943,A -85,B 0,C 180,E1 -22824.773,E2 -22824.773} C_VEL
LIN {X 0,Y 210.276,Z 469.521,A -85,B 0,C 180,E1 -22827.672,E2 -22827.672} C_VEL
LIN {X 0,Y 202.08,Z 471.023,A -85,B 0,C 180,E1 -22830.863,E2 -22830.863} C_VEL
LIN {X 0,Y 194.706,Z 471.474,A -85,B 0,C 180,E1 -22834.333,E2 -22834.333} C_VEL
LIN {X 0,Y 188.238,Z 470.835,A -85,B 0,C 180,E1 -22838.077,E2 -22838.077} C_VEL
LIN {X 0,Y 182.814,Z 469.042,A -85,B 0,C 180,E1 -22842.089,E2 -22842.089} C_VEL
LIN {X 0,Y 178.371,Z 466.068,A -85,B 0,C 180,E1 -22846.326,E2 -22846.326} C_VEL
LIN {X 0,Y 175.174,Z 461.834,A -85,B 0,C 180,E1 -22850.765,E2 -22850.765} C_VEL
LIN {X 0,Y 173.409,Z 457.76,A -85,B 0,C 180,E1 -22854.185,E2 -22854.185} C_VEL
LIN {X 0,Y 171.829,Z 451.109,A -85,B 0,C 180,E1 -22858.828,E2 -22858.828} C_VEL
LIN {X 0,Y 171.204,Z 443.919,A -85,B 0,C 180,E1 -22862.942,E2 -22862.942} C_VEL
LIN {X 0,Y 171.502,Z 433.937,A -85,B 0,C 180,E1 -22867.654,E2 -22867.654} C_VEL
LIN {X 0,Y 172.177,Z 425.676,A -85,B 0,C 180,E1 -22870.912,E2 -22870.912} C_VEL
LIN {X 0,Y 173.231,Z 416.3,A -85,B 0,C 180,E1 -22874.089,E2 -22874.089} C_VEL
LIN {X 0,Y 174.591,Z 404.101,A -85,B 0,C 180,E1 -22877.572,E2 -22877.572} C_VEL
LIN {X 0,Y 176.384,Z 390.7,A -85,B 0,C 180,E1 -22880.709,E2 -22880.709} C_VEL
LIN {X 0,Y 176.961,Z 386.762,A -85,B 0,C 180,E1 -22881.553,E2 -22881.553} C_VEL
LIN {X 0,Y 177.43,Z 387.193,A -85,B 0,C 180,E1 -22882.105,E2 -22882.105} C_VEL
LIN {X 0,Y 179.048,Z 386.068,A -85,B 0,C 180,E1 -22883.112,E2 -22883.112} C_VEL
LIN {X 0,Y 181.716,Z 382.709,A -85,B 0,C 180,E1 -22884.316,E2 -22884.316} C_VEL
LIN {X 0,Y 185.36,Z 376.704,A -85,B 0,C 180,E1 -22885.55,E2 -22885.55} C_VEL
LIN {X 0,Y 185.606,Z 376.417,A -85,B 0,C 180,E1 -22885.664,E2 -22885.664} C_VEL
LIN {X 0,Y 187.015,Z 375.915,A -85,B 0,C 180,E1 -22886.504,E2 -22886.504} C_VEL
LIN {X 0,Y 189.341,Z 373.648,A -85,B 0,C 180,E1 -22887.569,E2 -22887.569} C_VEL
LIN {X 0,Y 191.713,Z 370.535,A -85,B 0,C 180,E1 -22888.462,E2 -22888.462} C_VEL
LIN {X 0,Y 192.647,Z 369.867,A -85,B 0,C 180,E1 -22888.889,E2 -22888.889} C_VEL
LIN {X 0,Y 193.69,Z 369.949,A -85,B 0,C 180,E1 -22889.482,E2 -22889.482} C_VEL
LIN {X 0,Y 197.398,Z 375.418,A -85,B 0,C 180,E1 -22892.204,E2 -22892.204} C_VEL
LIN {X 0,Y 200.753,Z 381.164,A -85,B 0,C 180,E1 -22894.673,E2 -22894.673} C_VEL
LIN {X 0,Y 204.717,Z 389.983,A -85,B 0,C 180,E1 -22897.851,E2 -22897.851} C_VEL
LIN {X 0,Y 207.192,Z 397.101,A -85,B 0,C 180,E1 -22900.127,E2 -22900.127} C_VEL
LIN {X 0,Y 209.404,Z 407.9,A -85,B 0,C 180,E1 -22903.144,E2 -22903.144} C_VEL
LIN {X 0,Y 210.482,Z 417.9,A -85,B 0,C 180,E1 -22905.879,E2 -22905.879} C_VEL
LIN {X 0,Y 210.514,Z 419.214,A -85,B 0,C 180,E1 -22906.216,E2 -22906.216} C_VEL
LIN {X 0,Y 205.83,Z 431.248,A -85,B 0,C 180,E1 -22908.254,E2 -22908.254} C_VEL
LIN {X 0,Y 201.046,Z 442.133,A -85,B 0,C 180,E1 -22910.546,E2 -22910.546} C_VEL
LIN {X 0,Y 196.373,Z 452.07,A -85,B 0,C 180,E1 -22913.168,E2 -22913.168} C_VEL
LIN {X 0,Y 191.655,Z 460.959,A -85,B 0,C 180,E1 -22915.997,E2 -22915.997} C_VEL
LIN {X 0,Y 186.729,Z 469.651,A -85,B 0,C 180,E1 -22919.462,E2 -22919.462} C_VEL
LIN {X 0,Y 183.015,Z 475.872,A -85,B 0,C 180,E1 -22922.56,E2 -22922.56} C_VEL
LIN {X 0,Y 178.747,Z 482.736,A -85,B 0,C 180,E1 -22926.847,E2 -22926.847} C_VEL
LIN {X 0,Y 175.465,Z 488.103,A -85,B 0,C 180,E1 -22931.311,E2 -22931.311} C_VEL
LIN {X 0,Y 172.968,Z 492.153,A -85,B 0,C 180,E1 -22935.889,E2 -22935.889} C_VEL
LIN {X 0,Y 171.316,Z 494.981,A -85,B 0,C 180,E1 -22940.555,E2 -22940.555} C_VEL
LIN {X 0,Y 170.49,Z 496.66,A -85,B 0,C 180,E1 -22945.27,E2 -22945.27} C_VEL
LIN {X 0,Y 170.23,Z 497.238,A -85,B 0,C 180,E1 -22949.999,E2 -22949.999} C_VEL
LIN {X 0,Y 170.456,Z 496.691,A -85,B 0,C 180,E1 -22954.73,E2 -22954.73} C_VEL
LIN {X 0,Y 171.317,Z 495.048,A -85,B 0,C 180,E1 -22959.444,E2 -22959.444} C_VEL
LIN {X 0,Y 172.962,Z 492.265,A -85,B 0,C 180,E1 -22964.11,E2 -22964.11} C_VEL
LIN {X 0,Y 175.423,Z 488.269,A -85,B 0,C 180,E1 -22968.693,E2 -22968.693} C_VEL
LIN {X 0,Y 178.695,Z 482.945,A -85,B 0,C 180,E1 -22973.159,E2 -22973.159} C_VEL
LIN {X 0,Y 182.964,Z 476.126,A -85,B 0,C 180,E1 -22977.448,E2 -22977.448} C_VEL
LIN {X 0,Y 187.296,Z 468.812,A -85,B 0,C 180,E1 -22981.06,E2 -22981.06} C_VEL
LIN {X 0,Y 192.307,Z 459.969,A -85,B 0,C 180,E1 -22984.503,E2 -22984.503} C_VEL
LIN {X 0,Y 197.049,Z 450.908,A -85,B 0,C 180,E1 -22987.324,E2 -22987.324} C_VEL
LIN {X 0,Y 202.05,Z 440.137,A -85,B 0,C 180,E1 -22990.072,E2 -22990.072} C_VEL
LIN {X 0,Y 207.138,Z 428.423,A -85,B 0,C 180,E1 -22992.403,E2 -22992.403} C_VEL
LIN {X 0,Y 210.431,Z 419.731,A -85,B 0,C 180,E1 -22993.856,E2 -22993.856} C_VEL
LIN {X 0,Y 210.634,Z 418.34,A -85,B 0,C 180,E1 -22994.143,E2 -22994.143} C_VEL
LIN {X 0,Y 209.371,Z 407.303,A -85,B 0,C 180,E1 -22997.178,E2 -22997.178} C_VEL
LIN {X 0,Y 207.64,Z 398.803,A -85,B 0,C 180,E1 -22999.562,E2 -22999.562} C_VEL
LIN {X 0,Y 205.769,Z 392.701,A -85,B 0,C 180,E1 -23001.44,E2 -23001.44} C_VEL
LIN {X 0,Y 202.219,Z 384.127,A -85,B 0,C 180,E1 -23004.399,E2 -23004.399} C_VEL
LIN {X 0,Y 198.173,Z 376.519,A -85,B 0,C 180,E1 -23007.47,E2 -23007.47} C_VEL
LIN {X 0,Y 195.71,Z 372.391,A -85,B 0,C 180,E1 -23009.321,E2 -23009.321} C_VEL
LIN {X 0,Y 193.304,Z 368.566,A -85,B 0,C 180,E1 -23011.2,E2 -23011.2} C_VEL
LIN {X 0,Y 190.698,Z 364.763,A -85,B 0,C 180,E1 -23013.243,E2 -23013.243} C_VEL
LIN {X 0,Y 187.39,Z 360.555,A -85,B 0,C 180,E1 -23016.003,E2 -23016.003} C_VEL
LIN {X 0,Y 186.442,Z 359.262,A -85,B 0,C 180,E1 -23016.846,E2 -23016.846} C_VEL
LIN {X 0,Y 183.217,Z 355.476,A -85,B 0,C 180,E1 -23019.95,E2 -23019.95} C_VEL
LIN {X 0,Y 182.359,Z 354.233,A -85,B 0,C 180,E1 -23020.878,E2 -23020.878} C_VEL
LIN {X 0,Y 179.35,Z 351.572,A -85,B 0,C 180,E1 -23024.371,E2 -23024.371} C_VEL
LIN {X 0,Y 177.915,Z 349.278,A -85,B 0,C 180,E1 -23026.726,E2 -23026.726} C_VEL
LIN {X 0,Y 178.088,Z 348.549,A -85,B 0,C 180,E1 -23030.917,E2 -23030.917} C_VEL
LIN {X 0,Y 178.228,Z 348.439,A -85,B 0,C 180,E1 -23035.476,E2 -23035.476} C_VEL
LIN {X 0,Y 178.869,Z 348.543,A -85,B 0,C 180,E1 -23040,E2 -23040} C_VEL
LIN {X 0,Y 179.053,Z 349.708,A -85,B 0,C 180,E1 -23044.502,E2 -23044.502} C_VEL
LIN {X 0,Y 179.764,Z 351.234,A -85,B 0,C 180,E1 -23048.997,E2 -23048.997} C_VEL
LIN {X 0,Y 180.488,Z 353.513,A -85,B 0,C 180,E1 -23053.511,E2 -23053.511} C_VEL
LIN {X 0,Y 181.729,Z 356.453,A -85,B 0,C 180,E1 -23057.876,E2 -23057.876} C_VEL
LIN {X 0,Y 186.105,Z 362.548,A -85,B 0,C 180,E1 -23062.187,E2 -23062.187} C_VEL
LIN {X 0,Y 188.04,Z 364.75,A -85,B 0,C 180,E1 -23063.762,E2 -23063.762} C_VEL
LIN {X 0,Y 192.418,Z 371.3,A -85,B 0,C 180,E1 -23067.091,E2 -23067.091} C_VEL
LIN {X 0,Y 195.837,Z 378.002,A -85,B 0,C 180,E1 -23069.567,E2 -23069.567} C_VEL
LIN {X 0,Y 200.684,Z 388.081,A -85,B 0,C 180,E1 -23072.949,E2 -23072.949} C_VEL
LIN {X 0,Y 205.044,Z 399.103,A -85,B 0,C 180,E1 -23076.094,E2 -23076.094} C_VEL
LIN {X 0,Y 208.774,Z 409.98,A -85,B 0,C 180,E1 -23078.95,E2 -23078.95} C_VEL
LIN {X 0,Y 208.965,Z 412.594,A -85,B 0,C 180,E1 -23079.437,E2 -23079.437} C_VEL
LIN {X 0,Y 208.208,Z 424.525,A -85,B 0,C 180,E1 -23081.279,E2 -23081.279} C_VEL
LIN {X 0,Y 206.113,Z 438.681,A -85,B 0,C 180,E1 -23083.62,E2 -23083.62} C_VEL
LIN {X 0,Y 203.185,Z 452.384,A -85,B 0,C 180,E1 -23086.229,E2 -23086.229} C_VEL
LIN {X 0,Y 202.192,Z 455.604,A -85,B 0,C 180,E1 -23086.881,E2 -23086.881} C_VEL
LIN {X 0,Y 196.752,Z 467.783,A -85,B 0,C 180,E1 -23089.316,E2 -23089.316} C_VEL
LIN {X 0,Y 191.303,Z 478.606,A -85,B 0,C 180,E1 -23092.023,E2 -23092.023} C_VEL
LIN {X 0,Y 185.788,Z 489.193,A -85,B 0,C 180,E1 -23095.43,E2 -23095.43} C_VEL
LIN {X 0,Y 181.034,Z 497.984,A -85,B 0,C 180,E1 -23099.027,E2 -23099.027} C_VEL
LIN {X 0,Y 177.102,Z 505.392,A -85,B 0,C 180,E1 -23102.848,E2 -23102.848} C_VEL
LIN {X 0,Y 173.53,Z 512.254,A -85,B 0,C 180,E1 -23107.372,E2 -23107.372} C_VEL
LIN {X 0,Y 171.117,Z 517.665,A -85,B 0,C 180,E1 -23112.06,E2 -23112.06} C_VEL
LIN {X 0,Y 169.999,Z 520.805,A -85,B 0,C 180,E1 -23115.638,E2 -23115.638} C_VEL
LIN {X 0,Y 169.45,Z 523.59,A -85,B 0,C 180,E1 -23119.875,E2 -23119.875} C_VEL
LIN {X 0,Y 168.863,Z 524.588,A -85,B 0,C 180,E1 -23121.834,E2 -23121.834} C_VEL
LIN {X 0,Y 167.529,Z 525.288,A -85,B 0,C 180,E1 -23123.789,E2 -23123.789} C_VEL
LIN {X 0,Y 164.278,Z 525.923,A -85,B 0,C 180,E1 -23127.773,E2 -23127.773} C_VEL
LIN {X 0,Y 163.018,Z 525.868,A -85,B 0,C 180,E1 -23130.545,E2 -23130.545} C_VEL
LIN {X 0,Y 162.636,Z 525.217,A -85,B 0,C 180,E1 -23134.959,E2 -23134.959} C_VEL
LIN {X 0,Y 162.376,Z 523.284,A -85,B 0,C 180,E1 -23139.97,E2 -23139.97} C_VEL
LIN {X 0,Y 163.061,Z 520.141,A -85,B 0,C 180,E1 -23144.988,E2 -23144.988} C_VEL
LIN {X 0,Y 164.832,Z 515.733,A -85,B 0,C 180,E1 -23149.944,E2 -23149.944} C_VEL
LIN {X 0,Y 167.737,Z 509.965,A -85,B 0,C 180,E1 -23154.771,E2 -23154.771} C_VEL
LIN {X 0,Y 171.907,Z 502.699,A -85,B 0,C 180,E1 -23159.38,E2 -23159.38} C_VEL
LIN {X 0,Y 175.885,Z 495.61,A -85,B 0,C 180,E1 -23162.953,E2 -23162.953} C_VEL
LIN {X 0,Y 177.798,Z 492.523,A -85,B 0,C 180,E1 -23164.283,E2 -23164.283} C_VEL
LIN {X 0,Y 187.301,Z 487.573,A -85,B 0,C 180,E1 -23169.635,E2 -23169.635} C_VEL
LIN {X 0,Y 197.776,Z 481.961,A -85,B 0,C 180,E1 -23173.864,E2 -23173.864} C_VEL
LIN {X 0,Y 207.309,Z 476.692,A -85,B 0,C 180,E1 -23176.793,E2 -23176.793} C_VEL
LIN {X 0,Y 222.37,Z 467.711,A -85,B 0,C 180,E1 -23180.443,E2 -23180.443} C_VEL
LIN {X 0,Y 223.847,Z 466.571,A -85,B 0,C 180,E1 -23181.103,E2 -23181.103} C_VEL
LIN {X 0,Y 213.913,Z 469.717,A -85,B 0,C 180,E1 -23183.745,E2 -23183.745} C_VEL
LIN {X 0,Y 204.6,Z 471.868,A -85,B 0,C 180,E1 -23186.661,E2 -23186.661} C_VEL
LIN {X 0,Y 196.118,Z 472.965,A -85,B 0,C 180,E1 -23189.888,E2 -23189.888} C_VEL
LIN {X 0,Y 188.492,Z 473.025,A -85,B 0,C 180,E1 -23193.422,E2 -23193.422} C_VEL
LIN {X 0,Y 181.771,Z 472.016,A -85,B 0,C 180,E1 -23197.255,E2 -23197.255} C_VEL
LIN {X 0,Y 176.117,Z 469.866,A -85,B 0,C 180,E1 -23201.383,E2 -23201.383} C_VEL
LIN {X 0,Y 171.511,Z 466.533,A -85,B 0,C 180,E1 -23205.767,E2 -23205.767} C_VEL
LIN {X 0,Y 168.195,Z 461.954,A -85,B 0,C 180,E1 -23210.379,E2 -23210.379} C_VEL
LIN {X 0,Y 165.803,Z 456.051,A -85,B 0,C 180,E1 -23215.137,E2 -23215.137} C_VEL
LIN {X 0,Y 164.482,Z 448.648,A -85,B 0,C 180,E1 -23220,E2 -23220} C_VEL
LIN {X 0,Y 164.138,Z 440.756,A -85,B 0,C 180,E1 -23224.298,E2 -23224.298} C_VEL
LIN {X 0,Y 164.659,Z 431.298,A -85,B 0,C 180,E1 -23228.592,E2 -23228.592} C_VEL
LIN {X 0,Y 165.765,Z 419.545,A -85,B 0,C 180,E1 -23233.032,E2 -23233.032} C_VEL
LIN {X 0,Y 167.13,Z 407.301,A -85,B 0,C 180,E1 -23236.804,E2 -23236.804} C_VEL
LIN {X 0,Y 167.771,Z 401.945,A -85,B 0,C 180,E1 -23238.312,E2 -23238.312} C_VEL
LIN {X 0,Y 168.766,Z 401.992,A -85,B 0,C 180,E1 -23239.46,E2 -23239.46} C_VEL
